# B&R Automation Studio project Soiled_PLC (part 13)

#### empty.var - Local variables
```iecst
(********************************************************************
 * COPYRIGHT --
 ********************************************************************
 * Program: pr
 * File: pr.var
 * Author: treamsbottom
 * Created: July 16, 2015
 ********************************************************************
 * Local variables of program pr
 ********************************************************************)
VAR
	mySeq : UINT;
	myIO : UINT;
	myZone : UINT;
	myRelLine : UINT;
	myBag : UINT;
	i_bagAtBuffer : BOOL;
	i_bagAtBufferOut : BOOL;
	i_bufferOutOpen : BOOL;
	o_openBuffer : BOOL;
	step : UINT;
	pls : BOOL;
	timerAlarm : TON_10ms;
END_VAR
VAR RETAIN
	lastStep : UINT;
END_VAR
VAR
	bufferSettleTime : UDINT;
	myOutBag : UINT;
	myBuffBag : UINT;
	myCan : UINT;
	alarm : REFERENCE TO Alm;
	bag : REFERENCE TO Bag_typ;
	bag_buff : REFERENCE TO Bag_typ;
	bag_out : REFERENCE TO Bag_typ;
	can : REFERENCE TO CAN_Vars;
	line_release : REFERENCE TO Line_Typ;
END_VAR
```

### Package Logical/BaseStandards/Incline - *Incline conveyor

- Standard_Sequence_Incline_ENG.docx (binary file, 206111 bytes)
### Program Logical/BaseStandards/Incline/ic (IEC, version 1.00.5) - *incline

#### ic.st - Implementation code
```iecst
(********************************************************************
 * COPYRIGHT --
 ********************************************************************
 * Program: ic
 * File: ic.st
 * Author: treamsbottom
 * Created: July 17, 2015
 ********************************************************************
 * Implementation of program Incline conveyor.
 ********************************************************************)
//V1.00.1 First Release
PROGRAM _INIT
//Configuration
mySeq					:= 15;		//Sequence number
myIO					:= 171; 	//Incline Conveyor IO module number
myIC					:= 1;		//Incline Conveyor Number
useRequest				:= FALSE; 	//Use the Request bit. Only use when working with x_1_point. otherwise use RequestRelease as the i_bagAtBuffer.
myBuffBag				:= 270;		//Ingoing Buffer bag number
myBag					:= 290;		//Incline bag number
myRelLine				:= 23;
myOutBag				:= Line[myRelLine].LastBag;	//Outgoing buffer bag number

myZone 					:= 0;
//Timer Values
bufferSettleTime		:= 300;  	// Time for bag to settle at buffer in.
moveUpInclineTime		:= 8;//>>IN SECONDS<< // Time to move bag up incline after closing stop.//Min of 4 to shut buffer stop....

alarm						ACCESS ADR(Alarm[mySeq]);
bag							ACCESS ADR(Bag[myBag]);
bag_buff					ACCESS ADR(Bag[myBuffBag]);
bag_out						ACCESS ADR(Bag[myOutBag]);
line_release				ACCESS ADR(Line[myRelLine]);
END_PROGRAM

PROGRAM _CYCLIC
//Inputs
i_paddleInPosition		:= X[myIO].X01;
i_bagAtBuffer			:= X[myIO].X03;
i_bagInIncline			:= X[myIO].X04;
i_BagReleased			:= FALSE;//X[myIO].X05;  //<--- Bag release trip- only to be used in special cases. Take when using tracked bags, as the next sequence will need to copy data into a transit position

i_bagAtBufferOut 		:= FALSE; // Any Single bag buffer out IO.
i_bufferOutOpen			:= FALSE;

//End of inputs.

o_openBuffer			:= FALSE;
o_runMotor				:= FALSE;

Request.IC[myIC] 		:= FALSE;
RequestRel.IC[myIC] 	:= FALSE;

IF (myBag = 0) THEN
	alarm.Bag	:= mySeq + 10000;
ELSE
	alarm.Bag	:= myBag;
END_IF;

alarm.Name 		:= 0;
alarm.Beacon		:= TRUE;
alarm.Extra		:= 0;
alarm.Time		:= 3000;

//Setup Sequence
step := D[900 + mySeq];
//Setup Pulse contact
pls := (step <> laststep);
laststep := step;

//Sequence
IF (step = 0) THEN
	//Disabled
END_IF;

//Run Incline until paddle in position
IF (step = 1) THEN
	o_runMotor := NOT i_paddleInPosition;
	IF i_paddleInPosition THEN
		D[900 + mySeq] := 2;
		Count[mySeq] := Count[mySeq] + 1;
	END_IF;
	IF NOT Std.HaltSysZone[myZone] THEN
		alarm.Name := ALM_SWITCH_FAULT;
	END_IF;
END_IF;

//Wait for at buffer
ton_10ms_SettledBuffer(IN:= i_bagAtBuffer, PT:= bufferSettleTime);
IF (step = 2) THEN
	IF NOT i_bagInIncline THEN
		IF useRequest THEN
			D[900 + mySeq] := 3;
		ELSE
			IF ton_10ms_SettledBuffer.Q THEN
				IF (myBuffBag > 0) THEN
					IF (bag_buff.Cat > 0) AND (bag.Cat = 0) THEN
						D[900 + mySeq] := 3;
					ELSIF (bag_buff.Cat = 0) THEN
						alarm.Name := ALM_BAG_DATA_ERROR;
						alarm.Bag := myBuffBag;
					ELSE
						alarm.Name := ALM_BAG_DATA_ERROR;
					END_IF;
				ELSE
					D[900 + mySeq] := 3;
				END_IF;
			ELSIF (myBuffBag > 0) AND (bag_buff.Cat > 0) THEN
				alarm.Name := ALM_BAG_NOT_SETTLED;
			END_IF;
		END_IF;
	ELSE
		alarm.Name := ALM_SWITCH_FAULT;
	END_IF;
END_IF;

//Open Buffer stop
IF (step = 3) THEN
	releaseValid := ((myBag = 0) OR ((bag.Cat = 0) AND (bag_buff.Cat > 0)));
	o_openBuffer	   := releaseValid AND NOT useRequest;
	Request.IC[myIC]  := releaseValid AND useRequest;
	IF i_bagInIncline AND releaseValid THEN
		IF (myBag > 0) THEN
			bag := bag_buff; //Clear empty buffer bag data if used
			bag_buff := Bag[0];
		END_IF;
		D[900 + mySeq] := 4;
	ELSIF (myBag > 0) THEN
		IF (bag.Cat > 0) THEN
			alarm.Name := ALM_BAG_DATA_ERROR;
			alarm.Time := 0;
		ELSIF (bag_buff.Cat = 0) THEN
			alarm.Name := ALM_BAG_DATA_ERROR;
			alarm.Bag := myBuffBag;
			alarm.Time := 0;
		ELSE
			alarm.Name  := ALM_BAG_NOT_ARRIVED;
		END_IF;
	ELSE
		alarm.Name  := ALM_BAG_NOT_ARRIVED;
	END_IF;
END_IF;

ton_10ms_SettledIncline(IN:= (step = 4), PT:= 300);
IF (step = 4) THEN
	o_openBuffer := NOT useRequest;
	IF ton_10ms_SettledIncline.Q THEN
		D[900 + mySeq] := 5;
	END_IF;
END_IF;

//Move Bag up incline
ctu_moveUpIncline(CU:=(step = 5) AND NOT Std.HaltSysZone[myZone] AND Std.Clock1s, RESET := (step <> 5), PV := moveUpInclineTime);
IF (step = 5) THEN
	o_openBuffer 	:= (ctu_moveUpIncline.CV <= 4) AND NOT useRequest;//Close buffer stop after 3 seconds running..
	o_runMotor 		:= TRUE;
	IF ctu_moveUpIncline.Q THEN
		D[900 + mySeq] := 6;
	ELSIF NOT Std.HaltSysZone[myZone] THEN
		alarm.Name := ALM_SWITCH_FAULT;
	END_IF;

END_IF;

//Check for line space.
IF (step = 6) THEN
	releaseValid := (NOT i_bagAtBufferOut AND NOT i_bufferOutOpen AND NOT i_BagReleased AND ((myBag = 0) OR ((bag.Cat > 0) AND (bag_out.Cat = 0))));
	IF (myRelLine > 0) THEN
		IF (line_release.Clear AND releaseValid) THEN
			C[myRelLine] := 0;
			D[900 + mySeq] := 7;
		END_IF;
		IF (line_release.Clear AND i_bagAtBufferOut) THEN
			alarm.Name := ALM_SWITCH_FAULT;
		ELSIF (myBag > 0) AND (bag.Cat = 0) THEN
			alarm.Name := ALM_BAG_DATA_ERROR;
			alarm.Time := 0;
		ELSIF line_release.Clear AND (myOutBag > 0) AND (bag_out.Cat > 0) THEN
			alarm.Name := ALM_BAG_DATA_ERROR;
			alarm.Bag := myOutBag;
			alarm.Time := 0;
		END_IF;
	ELSE
		RequestRel.IC[myIC] := releaseValid;
		IF EnableRel.IC[myIC] AND releaseValid THEN

			D[900 + mySeq] := 7;
		ELSIF (myBag > 0) AND (bag.Cat = 0) THEN
			alarm.Name := ALM_BAG_DATA_ERROR;
			alarm.Time := 0;
		ELSIF (myOutBag > 0) AND (bag_out.Cat > 0) THEN
			alarm.Name := ALM_BAG_DATA_ERROR;
			alarm.Bag := myOutBag;
			alarm.Time := 0;
		END_IF;
	END_IF;
	IF i_BagReleased THEN
		alarm.Name := ALM_SWITCH_FAULT;
		alarm.Time := 0;
	END_IF;
	releaseValid := 0; //Clear this as we are using it as a latch in line 7
END_IF;

//Run motor to release bag.
IF (step = 7) THEN
	IF (NOT i_bagAtBufferOut AND NOT i_bufferOutOpen AND ((myBag = 0) OR ((bag.Cat > 0) AND (bag_out.Cat = 0)))) THEN
		releaseValid := 1;
	END_IF;
	o_runMotor := releaseValid AND NOT Std.HaltSysZone[myZone];
	IF releaseValid THEN
		IF (myBag = 0) THEN
			IF (myRelLine > 0) THEN
				IF line_release.Trip THEN
					D[900 + mySeq] := 1;
				END_IF;
			ELSE
				IF NOT EnableRel.IC[myIC] OR i_BagReleased THEN
					D[900 + mySeq] := 1;
				END_IF;
			END_IF;
			IF NOT Std.HaltSysZone[myZone] THEN
				alarm.Name := ALM_BAG_NOT_RELEASED;
			END_IF;
		ELSE//Use tracking
			IF (myRelLine > 0) THEN
				IF line_release.Trip THEN
					bag_out := bag;
					bag := Bag[0];
					D[900 + mySeq] := 1;
				END_IF;
			ELSE
				IF (i_BagReleased OR NOT EnableRel.IC[myIC]) AND (bag.Cat = 0)  THEN // Make sure data is copied out by enabling sequence.
					D[900 + mySeq] := 1;
				ELSIF NOT EnableRel.IC[myIC] AND (bag.Cat > 0) THEN
					alarm.Name := ALM_BAG_DATA_ERROR;
				END_IF;
			END_IF;
		END_IF;
	ELSIF i_bagAtBufferOut OR i_bufferOutOpen THEN
			alarm.Name := ALM_SWITCH_FAULT;
			alarm.Time := 0;
	ELSIF (myBag > 0) THEN
		IF (bag.Cat = 0) THEN
			alarm.Name := ALM_BAG_DATA_ERROR;
			alarm.Time := 0;
		ELSIF (bag_out.Cat > 0) THEN
			alarm.Name := ALM_BAG_DATA_ERROR;
			alarm.Bag := myOutBag;
			alarm.Time := 0;
		END_IF;
	END_IF;
END_IF;

//-----------------------------------
//PLC Outputs - adjust TO suit system
//-----------------------------------

Y[7].Y01	:= o_runMotor;
Y[myIO].Y06 := o_openBuffer;

//Alarms
timerAlarm(IN := NOT pls AND (alarm.Name > 0),PT:= alarm.Time);

alarm.On 	:= timerAlarm.Q;
alarm.ET 	:= timerAlarm.ET;;

END_PROGRAM
```

### Package Logical/BaseStandards/LoadingUnit - *Loading Unit

- Standard_Sequence_IoadingUnit_ENG.docx (binary file, 208000 bytes)
### Program Logical/BaseStandards/LoadingUnit/lu (IEC, version 1.01.1) - *Loading Unit

#### lu.var - Local variables
```iecst
(********************************************************************
 * COPYRIGHT --
 ********************************************************************
 * Program: lu
 * File: lu.var
 * Author: treamsbottom
 * Created: July 17, 2015
 ********************************************************************
 * Local variables of program lu
 ********************************************************************)
VAR
	useRequest : BOOL;
	useCompressor : BOOL;
	ton_10ms_SteadyDown : TON_10ms;
	ton_10ms_SettleInLU : TON_10ms;
	timerAlarm : TON_10ms;
	switchFault : BOOL;
	step : UINT;
	releaseValid : BOOL;
	pls : BOOL;
	o_steadyCylinders : BOOL;
	o_openBuffer : BOOL;
	o_openBackStop : BOOL;
	o_moveCompressorDown : BOOL;
	myZone : UINT;
	mySeq : UINT;
	myRelLine : UINT;
	myOutBag : UINT;
	myLU : UINT;
	myIO : UINT;
	myBuffBag : UINT;
	myBag : UINT;
	lu_Enabled : BOOL;
END_VAR
VAR RETAIN
	lastStep : UINT;
END_VAR
VAR
	i_compressorAtTop : ARRAY[0..2] OF BOOL;
	i_compress : BOOL;
	i_bufferOutOpen : BOOL;
	i_bagInLoadingUnit : BOOL;
	i_bagFrontPast : BOOL;
	i_bagAtBufferOut : BOOL;
	i_bagAtBuffer : BOOL;
	compressorUp : BOOL;
	compress : BOOL;
	bufferSettleTime : UINT;
	myReportStn : UINT;
	myBelt : UINT;
	myCan : UINT;
	unloadFinished : BOOL;
	ton_10ms_LuClear : TON_10ms;
	ton_10ms_SettledBuffer : TON_10ms;
	ton_10ms_CompressCheck : TON_10ms;
	ton_10ms_CompressDown : TON_10ms;
	ton_10ms_CompressorCheck : TON_10ms;
	myPrg : USINT;
	myCat : UDINT;
	myCus : UDINT;
	myWgt : UINT;
	myMis : UDINT;
	alarm : REFERENCE TO Alm;
	bag : REFERENCE TO Bag_typ;
	bag_out : REFERENCE TO Bag_typ;
	bag_buff : REFERENCE TO Bag_typ;
	can : REFERENCE TO CAN_Vars;
	line_release : REFERENCE TO Line_Typ;
END_VAR
```

### lu.st - Implementation code
```iecst
(********************************************************************
 * COPYRIGHT --
 ********************************************************************
 * Program: lu
 * File: lu.st
 * Author: treamsbottom
 * Created: July 17, 2015
 ********************************************************************
 * Implementation of program lu
 ********************************************************************)
//V1.00.1 First Release
PROGRAM _INIT
//Configuration
mySeq						:= 1;	//Sequence number
myIO						:= 21;	//First IO Block
myLU						:= 1;	// Loading unit number
myZone						:= 0;	// Safety Zone
myRelLine					:= 22; 	// Release Line - Set to 0 to Request Release
myBag						:= 255; //Buffer Bag
myBuffBag					:= 0; 	// Tracking Empty bag in...
useRequest					:= FALSE; 	//Use the Request bit. Only use when working with x_1_point. otherwise use RequestRelease as the i_bagAtBuffer.
bufferSettleTime			:= 300; // Time for bag to settle in buffer

useCompressor				:= FALSE;
myReportStn					:= 0;//myLU// Set Station index for reports. 0 = no report write.

myBelt						:= 1;	// Set if loaded by a belt
myCan						:= 0;	// Set if using Kanlink...

myOutBag					:= Line[myRelLine].LastBag;

alarm						ACCESS ADR(Alarm[mySeq]);
bag							ACCESS ADR(Bag[myBag]);
bag_buff					ACCESS ADR(Bag[myBuffBag]);
bag_out						ACCESS ADR(Bag[myOutBag]);
can							ACCESS ADR(CAN[myCan]);
line_release				ACCESS ADR(Line[myRelLine]);

END_PROGRAM

PROGRAM _CYCLIC
//Inputs
i_bagAtBuffer			:= X[myIO].X01;
i_bagFrontPast			:= X[myIO].X02;
i_bagInLoadingUnit		:= X[myIO].X03;
i_compressorAtTop[1]	:= TRUE; // Set to TRUE if there is no compressor
i_compressorAtTop[2]	:= TRUE;
i_compress				:= FALSE;

i_bagAtBufferOut 		:= FALSE; // Any Single bag buffer out IO.
i_bufferOutOpen			:= FALSE;

o_openBuffer			:= FALSE;
o_steadyCylinders		:= FALSE;
o_openBackStop	 		:= FALSE;
o_moveCompressorDown	:= FALSE;

Request.LU[myLU]		:= FALSE;
RequestRel.LU[myLU]		:= FALSE;
IF (myBelt > 0) THEN
	EnableRel.TransferBelt[myBelt] := FALSE;
END_IF;
IF (myCan > 0) THEN
	can.ReadyToLoad := FALSE;
END_IF

IF (myBag = 0) THEN
	alarm.Bag	:= mySeq + 10000;
ELSE
	alarm.Bag	:= myBag;
END_IF;

alarm.Name 		:= 0;
alarm.Beacon		:= TRUE;
alarm.Extra		:= 0;
alarm.Time		:= 3000;

//Setup Sequence
step := D[900 + mySeq];
//Setup Pulse contact
pls := (step <> lastStep);
lastStep := step;

//Get BagID
IF (bag.Cat > 0) AND (bag.Bid = 0) AND (BidStn > 0) THEN
	bag.Bid := BidStn;
	BidStn := 0;
END_IF;

//Sequence
IF (step = 0) THEN
	//Disabled
END_IF;

lu_Enabled	:= ((D[mySeq] > 0) AND NOT Std.HaltSysZone[myZone]);

//Check loading unit is clear.
switchFault 	:= (i_bagFrontPast OR i_bagInLoadingUnit);
compressorUp 	:= (i_compressorAtTop[1] AND i_compressorAtTop[2]);
ton_10ms_LuClear(IN:= compressorUp AND NOT switchFault,PT:= 200);
IF (step = 1) THEN
	IF (ton_10ms_LuClear.Q AND lu_Enabled) THEN
		D[900 + mySeq] := 2;
		Count[mySeq] := Count[mySeq] + 1;
	END_IF;
	IF (switchFault OR NOT compressorUp) THEN
		alarm.Name := ALM_SWITCH_FAULT;
	END_IF;
END_IF;

// Step 2 - Wait for bag at buffer if used
ton_10ms_SettledBuffer(IN:= i_bagAtBuffer, PT:= bufferSettleTime);
IF (step = 2) THEN
	IF useRequest THEN
		D[900 + mySeq] := 3;
	ELSE
		IF ton_10ms_SettledBuffer.Q THEN
			IF (myBuffBag > 0) THEN
				IF (bag_buff.Cat > 0) AND (bag.Cat = 0) THEN
					D[900 + mySeq] := 3;
				ELSIF (bag_buff.Cat = 0) THEN
					alarm.Name := ALM_BAG_DATA_ERROR;
					alarm.Bag := myBuffBag;
				ELSE
					alarm.Name := ALM_BAG_DATA_ERROR;
				END_IF;
			ELSE
				D[900 + mySeq] := 3;
			END_IF;
		ELSIF (myBuffBag > 0) AND (bag_buff.Cat > 0) THEN
			alarm.Name := ALM_BAG_NOT_SETTLED;
		END_IF;
	END_IF;
END_IF;

//Open buffer stop / Request bag
IF (step = 3) THEN
	releaseValid := ((myBuffBag = 0) OR ((bag.Cat = 0) AND (bag_buff.Cat > 0)));
	o_openBuffer := releaseValid AND NOT useRequest;
	o_openBackStop := TRUE;
	Request.LU[myLU]  := releaseValid AND useRequest;
	IF i_bagFrontPast AND releaseValid THEN
		IF (myBuffBag > 0) THEN
			bag := bag_buff; //Clear empty buffer bag data if used
			bag_buff := Bag[0];
		END_IF;
		D[900 + mySeq] := 4;
	ELSIF (myBuffBag > 0) THEN
		IF (bag.Cat > 0) THEN
			alarm.Name := ALM_BAG_DATA_ERROR;
			alarm.Time := 0;
		ELSIF (bag_buff.Cat = 0) THEN
			alarm.Name := ALM_BAG_DATA_ERROR;
			alarm.Bag := myBuffBag;
			alarm.Time := 0;
		ELSE
			alarm.Name  := ALM_BAG_NOT_ARRIVED;
		END_IF;
	ELSE
		alarm.Name  := ALM_BAG_NOT_ARRIVED;
	END_IF;
END_IF;

//Step 4 - Bag settles in loading unit
ton_10ms_SettleInLU(IN:= i_bagInLoadingUnit,PT:= 300);
IF (step = 4) THEN
	IF ton_10ms_SettleInLU.Q THEN
		D[900 + mySeq] := 5;
	END_IF;
	alarm.Name := ALM_BAG_NOT_SETTLED;
END_IF;

//Steady cylinders on from steps 5 - 8
o_steadyCylinders := ((step >= 5) AND (step <= 8));

//Move Steady Cylinders down and check bag data
ton_10ms_SteadyDown(IN:= (step = 5), PT:= 200);
IF (step = 5) THEN
	IF ton_10ms_SteadyDown.Q  THEN
		IF (myBuffBag = 0) THEN
			IF (bag.Cat = 0) THEN
				D[900 + mySeq] := 6;
			ELSE
				alarm.Name := ALM_BAG_DATA_ERROR;
				alarm.Time := 0;
			END_IF;
		ELSE
			IF (bag.Cat = Std.MaxCats) THEN
				D[900 + mySeq] := 6;
			ELSE
				alarm.Name := ALM_BAG_DATA_ERROR;
				alarm.Time := 0;
			END_IF;
		END_IF;
	END_IF;
END_IF;

//Step 6 Wait for bag to be loaded..
IF (step = 6) THEN
	EnableRel.TransferBelt[myBelt] 	:= (myBelt > 0);
	IF (myCan > 0) THEN// Kanlink interface.
		can.ReadyToLoad 		:= NOT unloadFinished;
		IF (can.Category > 0) AND NOT unloadFinished THEN
			myPrg := UINT_TO_USINT(can.Program);
			myCat := can.Category;
			myCus := can.Customer;
			myWgt := can.Weight;
			myMis := can.BatchID;
		END_IF;
		// Get Program code
		IF ((myPrg = 0) AND (myCat > 0) AND (D32[100 + 20 * (myLU - 1)] <> myCat)) THEN
			D32[100 + 20 * (myLU - 1)] := myCat;
		ELSIF (D32[101 + 20 * (myLU - 1)] = myCat) THEN
			myPrg := UDINT_TO_USINT(D32[102 + 20 * (myLU - 1)]);
		END_IF;
		IF can.UnloadFinished THEN
			unloadFinished := TRUE;
		END_IF;
		IF (unloadFinished AND (myCat > 0) AND (myPrg > 0)) THEN
			bag.Prg := myPrg;
			bag.Cat := myCat;
			bag.Cus := myCus;
			bag.Wgt := myWgt;
			bag.Mis := myMis;
		END_IF;
	END_IF;

	IF (bag.Cat > 0) AND (bag.Prg > 0) AND ((bag.Cat <> Std.MaxCats) OR (myBuffBag = 0)) THEN
		IF (myReportStn > 0) THEN
			IF (ReportLoading[myReportStn].Cat = 0) THEN
				ReportLoading[myReportStn].Prg := bag.Prg;
				ReportLoading[myReportStn].Cat := bag.Cat;
				ReportLoading[myReportStn].Cus := bag.Cus;
				ReportLoading[myReportStn].Wgt := bag.Wgt;
				ReportLoading[myReportStn].Cnt := 0;
				ReportLoading[myReportStn].Stn := myReportStn;
				ReportLoading[myReportStn].Mcn := 0;
				ReportLoading[myReportStn].Bid := bag.Mis;
				D[900 + mySeq] := 7;
			END_IF;
		ELSE
			D[900 + mySeq] := 7;
		END_IF;
	ELSIF (myCan > 0) AND unloadFinished THEN
		alarm.Name := ALM_BAG_DATA_ERROR;
	END_IF;
ELSE
	D32[100 + 20 * (myLU - 1)] := 0;
	unloadFinished := FALSE;
	can.ReadyToLoad := FALSE;
	can.Program := 0;
	can.Category := 0;
	can.Customer := 0;
	can.Weight := 0;
	can.BatchID := 0;
END_IF;

//Step 7 Check If compression is required
ton_10ms_CompressCheck(IN:=(step = 7),PT:= 30);
IF (step = 7) THEN
	IF useCompressor THEN
		IF i_compress THEN
			compress := TRUE;
		END_IF;
		IF ton_10ms_CompressCheck.Q THEN
			IF compress THEN
				D[900 + mySeq] := 8; // Compress
			ELSE
				D[900 + mySeq] := 9;	// Check compressor is OK
			END_IF;
		END_IF;
	ELSE
		D[900 + mySeq] := 9;
	END_IF;
ELSE
	compress := FALSE;
END_IF;

//Step 8 move linen compressor down.
ton_10ms_CompressDown(IN:=(step = 8),PT:= 500);
IF (step = 8) THEN
	IF useCompressor THEN
		IF ton_10ms_CompressDown.Q THEN
			D[900 + mySeq] := 9;
		END_IF;
	ELSE
		D[900 + mySeq] := 9;
	END_IF;
END_IF;

//step 9 check compressor status
ton_10ms_CompressorCheck(IN:=((i_compressorAtTop[1] AND i_compressorAtTop[2]) OR NOT useCompressor),PT:= 200);
IF (step = 9) THEN
	IF ton_10ms_CompressorCheck.Q  AND NOT Std.HaltSysZone[myZone] THEN
		D[900 + mySeq] := 10;
	END_IF;
	alarm.Name := ALM_SWITCH_FAULT;
END_IF;

//Check for line space.
IF (step = 10) THEN
	releaseValid := (NOT i_bagAtBufferOut AND NOT i_bufferOutOpen AND (bag.Cat > 0) AND (bag_out.Cat = 0));
	IF NOT Std.HaltSysZone[myZone] THEN
		IF (myRelLine > 0) THEN
			IF (line_release.Clear AND releaseValid) THEN
				C[myRelLine] := 0;
				D[900 + mySeq] := 11;
			END_IF;
			IF (line_release.Clear AND i_bagAtBufferOut) THEN
				alarm.Name := ALM_SWITCH_FAULT;
			ELSIF (bag.Cat = 0) THEN
				alarm.Name := ALM_BAG_DATA_ERROR;
				alarm.Time := 0;
			ELSIF line_release.Clear AND (bag_out.Cat > 0) THEN
				alarm.Name := ALM_BAG_DATA_ERROR;
				alarm.Bag := myOutBag;
				alarm.Time := 0;
			END_IF;
		ELSE
			RequestRel.LU[myLU] := releaseValid;
			IF EnableRel.LU[myLU] AND releaseValid THEN
				D[900 + mySeq] := 11;
			ELSIF (myBag > 0) AND (bag.Cat = 0) THEN
				alarm.Name := ALM_BAG_DATA_ERROR;
				alarm.Time := 0;
			ELSIF (myOutBag > 0) AND (bag_out.Cat > 0) THEN
				alarm.Name := ALM_BAG_DATA_ERROR;
				alarm.Bag := myOutBag;
				alarm.Time := 0;
			END_IF;
		END_IF;
	END_IF;
END_IF;

//Release bag.
IF (step = 11) THEN
	releaseValid 	:= (NOT i_bagAtBufferOut AND NOT i_bufferOutOpen AND (bag.Cat > 0) AND (bag_out.Cat = 0));
	o_openBackStop := releaseValid;
	IF releaseValid THEN
		IF (myRelLine > 0) THEN
			IF line_release.Trip THEN
				bag_out := bag;
				bag := Bag[0];
				D[900 + mySeq] := 1;
			END_IF;
		ELSE
			IF NOT EnableRel.LU[myLU] AND (bag.Cat = 0) THEN // Make sure data is copied out by enabling sequence.
				D[900 + mySeq] := 1;
			ELSIF NOT EnableRel.LU[myLU] AND (bag.Cat > 0) THEN
				alarm.Name := ALM_BAG_DATA_ERROR;
			END_IF;
		END_IF;
	ELSIF i_bagAtBufferOut OR i_bufferOutOpen THEN
		alarm.Name := ALM_SWITCH_FAULT;
		alarm.Time := 0;
	ELSIF (bag.Cat = 0) THEN
		alarm.Name := ALM_BAG_DATA_ERROR;
		alarm.Time := 0;
	ELSIF (bag_out.Cat > 0) THEN
		alarm.Name := ALM_BAG_DATA_ERROR;
		alarm.Bag := myOutBag;
		alarm.Time := 0;
	END_IF;
END_IF;

//-----------------------------------
//PLC Outputs - adjust TO suit system
//-----------------------------------

Y[myIO].Y05 		:= o_openBuffer;
Y[myIO].Y06 		:= o_openBackStop;
Y[myIO].Y07 		:= o_steadyCylinders;
//Y[myIO + 1].Y05 	:= o_moveCompressorDown;
//Y[myIO + 1].Y06 	:= o_moveCompressorDown;
Y[myIO + 1].Y07 	:= o_steadyCylinders; //Elephants foot

//Alarms
timerAlarm(IN := NOT pls AND (alarm.Name > 0),PT:= alarm.Time);

alarm.On 	:= timerAlarm.Q;
alarm.ET 	:= timerAlarm.ET;

END_PROGRAM
```

### Package Logical/BaseStandards/On_Offgoing - *Old style on and offgoing points

- SequenceExample.doc (binary file, 73216 bytes)
### Program Logical/BaseStandards/On_Offgoing/x_pn (IEC) - *Ongoing Sequence

#### x_pn.ab
```automation-basic
PROGRAM _CYCLIC

;--------------------------------------
;Sequence 4 - Ongoing To Storage D[900 + mySeq]
;--------------------------------------

;--------------------------------------------------------------------------------
;Revision 1.00 06/11/2009 D.J. First Issue - Automatic Line Allocation with Areas
;--------------------------------------------------------------------------------
mySeq 			= 4
myZone 			= 0
myTransitBag	= 208
myStartStop		= 100

IF (myStartStop >= 100) THEN
	myStartStop = myStartStop + 7600
ENDIF

;Inputs
OnGoingEnable 		= ((D[mySeq] > 0) AND NOT Std.HaltSysZone[myZone])

I_BagatBuffer[1]		= X[221].X02
I_BagatBuffer[2]		= FALSE
I_BagatBuffer[3]		= FALSE
I_BagatBuffer[4]		= FALSE

O_Reset 		  		= FALSE
O_OpenSelect[1]			= FALSE
O_OpenSelect[2]			= FALSE
O_OpenSelect[3]			= FALSE
O_OpenSelect[4]			= FALSE

O_OpenBuffer[1]			= FALSE
O_OpenBuffer[2]			= FALSE
O_OpenBuffer[3]			= FALSE
O_OpenBuffer[4]			= FALSE

MaxBuffers 			= 1 	;Set Max Buffers to search
MinLine				= 1 	;Set First Storage Line
MaxLine				= 10		;Set Last Storage Line
MaxDepth			= 7    ;Capacity of the longest line - used in search

Alarm[mySeq].Name 		= 0
Alarm[mySeq].Bag		= myTransitBag
Alarm[mySeq].Beacon		= TRUE
Alarm[mySeq].Extra	 	= 0
Alarm[mySeq].Time		= 6000

;Setup Sequence
;--------------
STEP = D[900 + mySeq]
;Setup Pulse contact
PLS = (STEP <> LASTSTEP)
LASTSTEP = STEP

;Step 0 - Disabled
IF (STEP = 0) THEN
	;Disabled
ENDIF

;Step 1 - Reset Ongoing Points
TON_10ms((STEP = 1),300,ResetPoints,ResetPointsET)
IF (STEP = 1) THEN
	Dest  	= 0
	Buff 	= 0
	O_Reset = TRUE
	IF (ResetPoints AND OnGoingEnable) THEN
		D[900 + mySeq] = 2
	ENDIF
ENDIF

;Bag Settles at each buffer
TON_10ms(I_BagatBuffer[1],300,SettledBuffer[1],SettledBufferET[1])
;TON_10ms(I_BagatBuffer[2],300,SettledBuffer[2],SettledBufferET[2])
;TON_10ms(I_BagatBuffer[3],300,SettledBuffer[3],SettledBufferET[3])

BufferBagNum[1]	    = 211
;BufferBagNum[2]	= 161
;BufferBagNum[3]	= myTransitBag

;Step 2 - Search for a valid Bag at one of the buffers
IF (STEP = 2) THEN

	Buff 	= 0
	Dest 	= 0

	IF OnGoingEnable THEN

		Alarm[mySeq].Name 	= almNoAlarm

		;Search only 1 buffer bag per scan/task
		Buffer = Buffer + 1
		IF Buffer > MaxBuffers THEN
			Buffer = 1
		ENDIF
		;Set Test Value for Monitoring
		IF TestBuffer > 0 THEN
			Buffer = TestBuffer
		ENDIF

		BufferBag		= BufferBagNum[Buffer]
		BufferSettled 	= SettledBuffer[Buffer]
		BufferPrg 		= Bag[BufferBag].Prg
		BufferCat		= Bag[BufferBag].Cat
		BufferCus		= Bag[BufferBag].Cus
		BufferDst 		= Bag[BufferBag].Dst

		IF (BufferSettled AND (BufferCat > 0) AND (BufferPrg > 0) AND (BufferPrg <= Std.MaxProg) AND (OnGoingEnable)) THEN

			;Manual Destination has been set?
			IF (BufferDst > 0) THEN

				n = BufferDst
				IF ((n >= MinLine) AND (n <= MaxLine) AND (Line[n].Space > 0) AND Line[n].Clear) THEN
					Dest 	= n
					Buff 	= Buffer
					D[900 + mySeq] 	= 3
				ELSE
					Alarm[mySeq].Name 	= almDestinationNotValid
					Alarm[mySeq].Bag	= BufferBag
				ENDIF

			ELSE IF Std.AutoLineAllocation THEN ;/BufferDst > 0

				;Search Each Storage Area
				AreaChoice[1] = D[3000 + BufferPrg]
				AreaChoice[2] = D[3100 + BufferPrg]
				AreaChoice[3] = D[3200 + BufferPrg]
				AreaChoice[4] = D[3300 + BufferPrg]

				LOOP Area = 1 TO 4 DO

					AreaStartLine 	= D[250 + AreaChoice[Area]]
					AreaEndLine 	= D[270 + AreaChoice[Area]]
					AreaValid		= ((AreaStartLine > 0) AND (AreaEndLine > 0) AND (AreaEndLine >= AreaStartLine))
					IF AreaValid THEN

						;Search for a line with the same program
						;---------------------------------------
						LOOP myLine = AreaStartLine TO AreaEndLine DO
							myLineValid = ((myLine >= MinLine) AND (myLine <= MaxLine))
							myLineUsed	= (D[myStartStop + myLine] > 0) ;Start / Stop On
							IF myLineValid AND myLineUsed THEN
								n 			= myLine
								SearchBag 	= (Line[n].LastBag - Line[n].Space)
								IF ((SearchBag >= Line[n].FirstBag) AND (Bag[SearchBag].Prg = BufferPrg) AND (Line[n].Space > 0) AND Line[n].Clear) THEN
									;Found line with a matching program
									Dest 	= n
								ENDIF ;/SearchBag
							ENDIF ;/myLineValid
							EXITIF (Dest <> 0)
						ENDLOOP ;/myLine loop

						;Search for an empty line
						;------------------------
						IF (Dest = 0) THEN
							LOOP myLine = AreaStartLine TO AreaEndLine DO
								myLineValid = ((myLine >= MinLine) AND (myLine <= MaxLine))
								myLineUsed	= (D[myStartStop + myLine] > 0) ;Start / Stop On
								IF myLineValid AND myLineUsed THEN
									n 			= myLine
									SearchBag 	= (Line[n].FirstBag)
									IF ((Bag[SearchBag].Prg = 0) AND (Line[n].Space > 0) AND Line[n].Clear) THEN
										;Found line with a matching program
										Dest 	= n
									ENDIF ;/SearchBag
								ENDIF ;/myLineValid
							EXITIF (Dest <> 0)
							ENDLOOP ;/myLine loop
						ENDIF ;/Dest = 0

						;Search for a line that already contains a bag with the same program starting at the back
						;----------------------------------------------------------------------------------------
						IF (Dest = 0) THEN
							LOOP myDepth = (MaxDepth - 2) DOWNTO 0 DO ;Don't search the last bag as the line would already be full!!
								LOOP myLine = AreaStartLine TO AreaEndLine DO
									myLineValid = ((myLine >= MinLine) AND (myLine <= MaxLine))
									myLineUsed	= (D[myStartStop + myLine] > 0) ;Start / Stop On
									IF myLineValid AND myLineUsed THEN
										n 			= myLine
										SearchBag 	= (Line[n].FirstBag + myDepth)
										IF ((Bag[SearchBag].Prg = BufferPrg) AND (Line[n].Space > 0) AND Line[n].Clear) THEN
											;Found line with a matching program
											FoundDepth 	= myDepth
											Dest 		= n
										ENDIF ;/SearchBag
									ENDIF ;/myLineValid
									EXITIF (Dest <> 0)
								ENDLOOP ;/myLine loop
								EXITIF (Dest <> 0)
							ENDLOOP ;/myDepgh
						ENDIF ;/Dest = 0

						;Search for line with the most space
						;-----------------------------------
						IF (Dest = 0) THEN
							mySpace = 0
							myFound	= 0
							LOOP myLine = AreaStartLine TO AreaEndLine DO
								myLineValid = ((myLine >= MinLine) AND (myLine <= MaxLine))
								myLineUsed	= (D[myStartStop + myLine] > 0) ;Start / Stop On
								IF myLineValid AND myLineUsed THEN
									n 			= myLine
									SearchBag 	= (Line[n].LastBag)
									IF ((Bag[SearchBag].Prg = 0) AND (Line[n].Space > mySpace) AND Line[n].Clear) THEN
										;Found line with a matching program
										myFound	= n
										mySpace = Line[n].Space
									ENDIF ;/SearchBag
								ENDIF ;/myLineValid
							ENDLOOP ;/myLine loop

							IF (myFound > 0) THEN
								Dest 	= myFound
							ENDIF

						ENDIF ;/Dest = 0

					ENDIF ;/Area Valid
					EXITIF (Dest <> 0)
				ENDLOOP ;/Area Loop

			ENDIF ;/BufferDst > 0

			;Destination line found!!
			IF (Dest <> 0) THEN
				Buff = Buffer
				IF (Bag[myTransitBag].Cat = 0) AND (Bag[BufferBagNum[Buff]].Cat > 0) THEN ;Bag in Transit
					Bag[BufferBagNum[Buff]].Dst = USINT(Dest)
					Bag[myTransitBag]	= Bag[BufferBagNum[Buff]]
					Bag[BufferBagNum[Buff]]	 	= Bag[0]
					C[Dest] = 0
					D[900 + mySeq] 	= 3 ; Open buffer
				ENDIF
			ELSE
				;Storage full!!
				;Do Nothing? Alarm?
				;Other Area?
			ENDIF

		ENDIF ;/BagSettled

		;Buffer Alarms
		IF (BufferPrg > 0) AND NOT BufferSettled THEN
			Alarm[mySeq].Name 	= almBagNotAtProx
			Alarm[mySeq].Bag	= BufferBag
		ELSE IF (BufferPrg = 0) AND BufferSettled THEN
			Alarm[mySeq].Name 	= almBagNotShownOnScreen
			Alarm[mySeq].Bag	= BufferBag
		ENDIF
	ENDIF
ENDIF

;Clear Line Selections
LOOP n = 1 TO Std.MaxLines DO
	LineSelect[n] = FALSE
ENDLOOP

;Step 3 - Select line / open buffer stop
IF (STEP = 3) THEN
	LineSelect[Dest] 	= TRUE
	O_OpenBuffer[Buff] = TRUE
	;Bag arrived on selected line
	IF Line[Dest].Trip THEN
		D32[498] 					= Bag[myTransitBag].Cus	;Set Customer for Customer FIFO
		Bag[myTransitBag].Dst 		= 0 		    ;Clear Destination
		Bag[Line[Dest].LastBag] 	= Bag[myTransitBag]
		Bag[myTransitBag] 			= Bag[0]
		D[900 + mySeq] 				= 1
	ENDIF
	Alarm[mySeq].Name = almBagNotArrived
ENDIF

;Alarms
TimerAlarm.IN = NOT PLS AND (Alarm[mySeq].Name > 0) AND (AlarmOld = Alarm[mySeq].Name)
TimerAlarm.PT = Alarm[mySeq].Time
TimerAlarm FUB TON_10ms()
Alarm[mySeq].On = TimerAlarm.Q
Alarm[mySeq].ET = TimerAlarm.ET

AlarmOld = Alarm[mySeq].Name ;Need to ensure alarm changes as may be multiple alarms on step 2

Y[221].Y06 = O_OpenBuffer[1]

;Outputs
Y[51].Y08 = O_Reset
Y[52].Y07 = O_Reset
Y[53].Y07 = O_Reset
Y[53].Y08 = O_Reset
Y[54].Y07 = O_Reset
Y[54].Y08 = O_Reset
Y[55].Y07 = O_Reset
Y[55].Y08 = O_Reset
Y[56].Y07 = O_Reset

Y[51].Y06 = LineSelect[2]
Y[52].Y05 = LineSelect[3]
Y[53].Y05 = LineSelect[4]
Y[53].Y06 = LineSelect[5]
Y[54].Y05 = LineSelect[6]
Y[54].Y06 = LineSelect[7]
Y[55].Y05 = LineSelect[8]
Y[55].Y06 = LineSelect[9]
Y[56].Y05 = LineSelect[10]

END_PROGRAM
```

### Program Logical/BaseStandards/On_Offgoing/x_pf (IEC) - *Offgoing Sequence

#### pf1.var
```iecst
VAR RETAIN
	LASTSTEP : UINT;
	SelectedBuffer : USINT;
	Destination : UINT;
	FoundLine : UINT;
END_VAR
VAR
	x : UINT;
	Line14_Valid : BOOL;
	LongestLine : UINT;
	O_Select : ARRAY[0..22] OF BOOL;
	LongestSTime : UINT;
	LineInList : ARRAY[0..98] OF BOOL;
	mySeq : UINT;
	RecircSpaces : UINT;
	O_Reset3way : BOOL;
	r : UINT;
	myRelLine : UINT;
	SettleTime : UINT;
	TransitBag : UINT;
	RecircValid : BOOL;
	TimerAlarm : TON_10ms;
	SDC6_Valid : BOOL;
	SDC5_Valid : BOOL;
	SDC7_Valid : BOOL;
	TestAtStop : BOOL;
	STEP : UINT;
	SDC3_Valid : BOOL;
	SearchDest : UINT;
	SDC4_Valid : BOOL;
	I_InclineBufferStopOpen : BOOL;
	ResetPointsET : TIME;
	ResetPoints : BOOL;
	OffGoingEnable : BOOL;
	SDC1_Valid : BOOL;
	SDC2_Valid : BOOL;
	PLS : BOOL;
	O_SDCBufferOpen : ARRAY[0..4] OF BOOL;
	O_Reset : BOOL;
	MaxLine : UINT;
	n : UINT;
	MinLine : UINT;
	BufferBag : ARRAY[0..9] OF UINT;
	LineSelect : ARRAY[0..30] OF BOOL;
	MaxBuffers : UINT;
	I_SDCBagAtBuffer : ARRAY[0..4] OF BOOL;
	I_BagAtIncline : BOOL;
	IncSettle : BOOL;
	LineSettle : ARRAY[0..30] OF BOOL;
	BestTime : UINT;
	BufferClear : ARRAY[0..9] OF BOOL;
	AlarmBagNotProx : BOOL;
	I_BagAtStop : ARRAY[0..30] OF BOOL;
	BagSettledTime : ARRAY[0..30] OF UINT;
	myZone : UINT;
END_VAR
```

#### pf1.ab
```automation-basic
PROGRAM _CYCLIC

;----------------------------------------
;Sequence 5 - SPF1 Offgoing Points D[900+mySeq]
;----------------------------------------

;Inputs
;------
mySeq			= 5
myRelLine 		= 26
TransitBag 		= 207
myZone			= 0

OffGoingEnable 		= ((D[mySeq] > 0) AND NOT Std.HaltSysZone[myZone])

I_SDCBagAtBuffer[1] = X[213].X01 ;Bag In Discharger
I_SDCBagAtBuffer[2] = FALSE ;Use for single bag buffer
I_SDCBagAtBuffer[3] = FALSE ;X[6].X13 ;Use for single bag buffer
I_SDCBagAtBuffer[4] = FALSE ;X[6].X13 ;Use for single bag buffer

O_SDCBufferOpen[1]  = Y[213].Y05 ;Use for single bag buffer
O_SDCBufferOpen[2]  = FALSE ;Use for single bag buffer
O_SDCBufferOpen[3]  = FALSE ;Y[6].Y16 ;Use for single bag buffer
O_SDCBufferOpen[4]  = FALSE ;Y[6].Y16 ;Use for single bag buffer

I_BagAtStop[1]	 	= X[71].X01 OR TestAtStop
I_BagAtStop[2] 		= X[71].X02 OR TestAtStop
I_BagAtStop[3] 		= X[72].X01 OR TestAtStop
I_BagAtStop[4] 		= X[72].X02 OR TestAtStop
I_BagAtStop[5] 		= X[73].X01 OR TestAtStop
I_BagAtStop[6]	 	= X[73].X02 OR TestAtStop
I_BagAtStop[7] 		= X[74].X01 OR TestAtStop
I_BagAtStop[8] 		= X[74].X02 OR TestAtStop
I_BagAtStop[9] 		= X[75].X01 OR TestAtStop
I_BagAtStop[10] 	= X[75].X02 OR TestAtStop

O_Reset 			= FALSE

;Buffer line configuration
;-------------------------
MaxBuffers			= 1
MinLine				= 1
MaxLine				= 10

BufferBag[1]		= 251 ;Last buffer bag number
;BufferBag[2]		= 373;Last buffer bag number
;BufferBag[3]		= 383 ;Last buffer bag number CDC3
;BufferBag[4]		= 192 ;Last buffer bag number CDC4
;BufferBag[5]		= 155 ;Last buffer bag number CDC 5
;BufferBag[6]		= 658 ;Last buffer bag number
;BufferBag[7]		= 664 ;Last buffer bag number
;RecircSpaces  		=(Line[20].Space + Line[24].Space + (Bag[190].Cat = 0) - DestCountSystem[30])

BufferClear[1] 		= ((D[6]> 0) AND (Line[31].SpaceBIT > 0) )
;BufferClear[2]		= ((Bag[Line[22].LastBag].Cat = 0) AND  (Line[22].SpaceBIT >= 1)); Empty bag buffer before CDC2
;BufferClear[3]		= ((Bag[Line[23].LastBag].Cat = 0) AND  (Line[23].SpaceBIT >= 1))
;BufferClear[4]		= (Bag[BufferBag[4]].Cat = 0) AND (RecircSpaces > 0) ;Recirc Valid
;BufferClear[5]		= ((Bag[BufferBag[5]].Cat = 0) AND (D[10] > 0) AND Request.DC[5] AND (Line[25].SpaceBIT >= 1))
;;BufferClear[6]		= (D[9] > 0) AND (Bag[BufferBag[6]].Cat = 0)
;BufferClear[7]		= (D[10] > 0) AND (Bag[BufferBag[7]].Cat = 0)

Uld[1].SDCReady 	= BufferClear[1]
Uld[2].SDCReady 	= FALSE
Uld[3].SDCReady		= FALSE
Uld[4].SDCReady 	= FALSE
;Uld[5].SDCReady 	= BufferClear[5]

Alarm[mySeq].Name 		= 0
Alarm[mySeq].Bag		= TransitBag
Alarm[mySeq].Beacon		= TRUE
Alarm[mySeq].Extra		= 0
Alarm[mySeq].Time		= 45000

;Setup Sequence
;--------------
STEP = D[900 + mySeq]
;Setup Pulse contact
PLS = (STEP <> LASTSTEP)
LASTSTEP = STEP

;Sequence Steps
;--------------
IF (STEP = 0) THEN
	;Disabled
ENDIF

;Step 1 - Reset Points
TON_10ms((STEP = 1),300,ResetPoints,ResetPointsET)
IF (STEP = 1) THEN
	O_Reset 	= TRUE
	FoundLine 	= 0
	Destination = 0
	IF (ResetPoints AND OffGoingEnable) THEN
		D[900+mySeq] = 2
	ENDIF
ENDIF

;Bags on storage line timers
R_TRIG(Std.Clock100ms,IncSettle)
AlarmBagNotProx 	= FALSE
AlarmBagNotProxLine = 0

LOOP n = MinLine TO MaxLine DO

	LineSettle[n]  = (I_BagAtStop[n] AND (Bag[Line[n].FirstBag].Cat > 0))
	IF IncSettle AND LineSettle[n] AND (BagSettledTime[n] < $FFFF) THEN
		BagSettledTime[n] = BagSettledTime[n] + 1
	ELSE IF NOT LineSettle[n] THEN
		BagSettledTime[n] = 0
		;If Bag has destiantion and not at stop then alarm
		IF (Bag[Line[n].FirstBag].Dst > 0) THEN
			Alarm[mySeq].Name	= almBagNotAtProx
			Alarm[mySeq].Bag	= Line[n].FirstBag
			Alarm[mySeq].Extra 	= n
		ENDIF
	ENDIF
		LongestSTime = 0
		LongestTime[n] = 0
ENDLOOP

LOOP n = MinLine TO MaxLine DO
	LineInList[n]  = FALSE
ENDLOOP

LOOP n = MinLine TO MaxLine DO
	LongestLine = 0
	LongestSTime = 0
	LOOP x = MinLine TO MaxLine DO
		IF (BagSettledTime[x] > LongestSTime) AND NOT LineInList[x] THEN ;(BagSettledTime[x] > BagSettledTime[n]) AND
			LongestSTime = BagSettledTime[x]
			LongestLine = x
		ENDIF
	ENDLOOP
	LineInList[LongestLine] = TRUE
	LongestTime[n] = LongestLine
ENDLOOP

;Buffer trip not correct alarms
LOOP n = 1 TO MaxBuffers DO
	IF (STEP = 2) AND BufferClear[n] AND NOT Uld[n].SDCReady THEN
		;Alarm[mySeq].Name 	= almSwitchFault - Not direct to buffers
		;Alarm[mySeq].Bag	= BufferBag[n]
	ENDIF
ENDLOOP

;Search for the bag with a valid destination that has been waiting the longest
IF STEP = 2 THEN

	FoundLine 	= 0
	Destination = 0
	BestTime 	= 0
	SettleTime = 30 ;3 seconds

	LOOP n = MinLine TO MaxLine DO
		IF ((BagSettledTime[n] > SettleTime) AND (BagSettledTime[n] > BestTime)) THEN
			SearchDest = Bag[Line[n].FirstBag].Dst

			SDC1_Valid  = (SearchDest = 31) AND Uld[1].SDCReady
			SDC2_Valid 	= (SearchDest = 32) AND Uld[2].SDCReady
			SDC3_Valid 	= (SearchDest = 33) AND Uld[3].SDCReady
			SDC4_Valid 	= (SearchDest = 34) AND Uld[4].SDCReady
;			SDC5_Valid 	= ((SearchDest = 35) AND Uld[5].SDCReady)
            ;SDC6_Valid 	= ((SearchDest = 36) AND Uld[6].SDCReady)
			;SDC7_Valid 	= ((SearchDest = 37) AND Uld[7].SDCReady)
			;RecircValid = ((SearchDest = 30) AND Line[20].Clear AND (Bag[Line[20].LastBag].Cat = 0))
			IF SDC1_Valid THEN
				FoundLine 	= n
				Destination = SearchDest
				BestTime 	= BagSettledTime[n]
			ENDIF
		ENDIF
	ENDLOOP

	IF ((FoundLine > 0) AND (Destination > 0) AND OffGoingEnable AND (Bag[TransitBag].Cat = 0)) THEN
		IF Line[myRelLine].Clear AND (Bag[Line[myRelLine].LastBag].Cat = 0) AND (Bag[TransitBag] .Cat = 0) AND NOT I_SDCBagAtBuffer[1] AND NOT O_SDCBufferOpen[1] THEN
			C[myRelLine] = 0
			D[900 + mySeq] = 3
		ENDIF
	ENDIF
ENDIF

;Step 3 - Select Line / Open Stop, Until Bag at correct destination
;Clear Line Selections
LOOP n = MinLine TO MaxLine DO
	LineSelect[n] = FALSE
ENDLOOP

IF (STEP = 3) THEN
	LineSelect[FoundLine] = TRUE
	IF (Destination >= 21) AND (Destination <= 21) THEN
		Uld[Destination - 20].DischargerStartLine = FoundLine ;Unloading Program
	ENDIF
	IF (Bag[TransitBag] .Cat = 0) AND (Bag[Line[FoundLine].FirstBag].Cat > 0)THEN
		IF PLS THEN
			Bag[TransitBag]  = Bag[Line[FoundLine].FirstBag]
			Bag[Line[FoundLine].FirstBag] 	= Bag[0]
		ENDIF
	ENDIF
	IF Line[myRelLine].Trip THEN
		Bag[Line[myRelLine].LastBag] = Bag[TransitBag]
		Bag[TransitBag] = Bag[0]
		D[900 + mySeq] = 1
	ENDIF
	Alarm[mySeq].Name	= almBagNotReleased
ENDIF

;Alarms
TimerAlarm.IN = NOT PLS AND (Alarm[mySeq].Name > 0)
TimerAlarm.PT = Alarm[mySeq].Time
TimerAlarm FUB TON_10ms()
Alarm[mySeq].On = TimerAlarm.Q
Alarm[mySeq].ET = TimerAlarm.ET

;Outputs
;-------

Y[71].Y07 = O_Reset
Y[71].Y08 = O_Reset
Y[72].Y07 = O_Reset
Y[72].Y08 = O_Reset
Y[73].Y07 = O_Reset
Y[73].Y08 = O_Reset
Y[74].Y07 = O_Reset
Y[74].Y08 = O_Reset
Y[75].Y07 = O_Reset
Y[75].Y08 = O_Reset

Y[71].Y05 = LineSelect[1]
Y[71].Y06 = LineSelect[2] OR LineSelect[1]
Y[71].Y03 = LineSelect[2]
Y[72].Y05 = LineSelect[3]
Y[72].Y06 = LineSelect[4]
Y[73].Y05 = LineSelect[5]
Y[73].Y06 = LineSelect[6]
Y[74].Y05 = LineSelect[7]
Y[74].Y06 = LineSelect[8]
Y[75].Y05 = LineSelect[9]
Y[75].Y06 = LineSelect[10]

END_PROGRAM
```

### Program Logical/BaseStandards/On_Offgoing/12_PN2 (IEC) - *Ongoing Sequence

#### x_pn.var
```iecst
VAR
	AlarmOld : UINT;
	Area : UINT;
	AreaChoice : ARRAY[0..4] OF UINT;
	AreaEndLine : UINT;
	AreaStartLine : UINT;
	AreaValid : BOOL;
END_VAR
VAR RETAIN
	Buff : UINT;
END_VAR
VAR
	Buffer : UINT;
	BufferBag : UINT;
	BufferBagNum : ARRAY[0..4] OF UINT;
	BufferCat : UDINT;
	BufferCus : UDINT;
	BufferDst : UINT;
	BufferPrg : UINT;
	BufferSettled : BOOL;
END_VAR
VAR RETAIN
	Dest : UINT;
END_VAR
VAR
	FoundDepth : UINT;
	I_BagatBuffer : ARRAY[0..4] OF BOOL;
END_VAR
VAR RETAIN
	LASTSTEP : UINT;
	LineSelect : ARRAY[0..19] OF BOOL;
END_VAR
VAR
	MaxBuffers : UINT;
	MaxDepth : UINT;
	MaxLine : UINT;
	MinLine : UINT;
	myDepth : UINT;
	myFound : UINT;
	myLine : UINT;
	myLineUsed : BOOL;
	myLineValid : BOOL;
	mySpace : UINT;
	n : UINT;
	O_OpenSelect : ARRAY[0..4] OF BOOL;
	O_Reset : BOOL;
	OnGoingEnable : BOOL;
END_VAR
VAR RETAIN
	PLS : BOOL;
END_VAR
VAR
	ResetPoints : BOOL;
	ResetPointsET : TIME;
	SearchBag : UINT;
	SettledBuffer : ARRAY[0..4] OF BOOL;
	SettledBufferET : ARRAY[0..4] OF TIME;
END_VAR
VAR RETAIN
	STEP : UINT;
END_VAR
VAR
	TestBuffer : UINT;
	TimerAlarm : TON_10ms;
	I_BagBagReleased : BOOL;
	mySeq : UINT;
	myZone : UINT;
	myTransitBag : UINT;
	myStartStop : UINT;
	O_OpenBuffer : ARRAY[0..9] OF BOOL;
END_VAR
```

#### x_pn.ab
```automation-basic
PROGRAM _CYCLIC

;--------------------------------------
;Sequence 4 - Ongoing To Storage D[900 + mySeq]
;--------------------------------------

;--------------------------------------------------------------------------------
;Revision 1.00 06/11/2009 D.J. First Issue - Automatic Line Allocation with Areas
;--------------------------------------------------------------------------------
mySeq 			= 4
myZone 			= 0
myTransitBag	= 298
myStartStop		= 100

IF (myStartStop >= 100) THEN
	myStartStop = myStartStop + 7600
ENDIF

;Inputs
OnGoingEnable 		= ((D[mySeq] > 0) AND NOT Std.HaltSysZone[myZone])

I_BagatBuffer[1]		= Request.VC[2]
I_BagatBuffer[2]		= FALSE
I_BagatBuffer[3]		= FALSE
I_BagatBuffer[4]		= FALSE

O_Reset 		  		= FALSE
O_OpenSelect[1]			= FALSE
O_OpenSelect[2]			= FALSE
O_OpenSelect[3]			= FALSE
O_OpenSelect[4]			= FALSE

O_OpenBuffer[1]			= FALSE
O_OpenBuffer[2]			= FALSE
O_OpenBuffer[3]			= FALSE
O_OpenBuffer[4]			= FALSE

MaxBuffers 			= 1 	;Set Max Buffers to search
MinLine				= 6 	;Set First Storage Line
MaxLine				= 11		;Set Last Storage Line
MaxDepth			= 9    ;Capacity of the longest line - used in search

Alarm[mySeq].Name 		= 0
Alarm[mySeq].Bag		= myTransitBag
Alarm[mySeq].Beacon		= TRUE
Alarm[mySeq].Extra	 	= 0
Alarm[mySeq].Time		= 6000

;Setup Sequence
;--------------
STEP = D[900 + mySeq]
;Setup Pulse contact
PLS = (STEP <> LASTSTEP)
LASTSTEP = STEP

;Step 0 - Disabled
IF (STEP = 0) THEN
	;Disabled
ENDIF

;Step 1 - Reset Ongoing Points
TON_10ms((STEP = 1),300,ResetPoints,ResetPointsET)
IF (STEP = 1) THEN
	Dest  	= 0
	Buff 	= 0
	O_Reset = TRUE
	IF (ResetPoints AND OnGoingEnable) THEN
		D[900 + mySeq] = 2
	ENDIF
ENDIF

;Bag Settles at each buffer
TON_10ms(I_BagatBuffer[1],300,SettledBuffer[1],SettledBufferET[1])
;TON_10ms(I_BagatBuffer[2],300,SettledBuffer[2],SettledBufferET[2])
;TON_10ms(I_BagatBuffer[3],300,SettledBuffer[3],SettledBufferET[3])

BufferBagNum[1]	    = 296
;BufferBagNum[2]	= 161
;BufferBagNum[3]	= myTransitBag

;Step 2 - Search for a valid Bag at one of the buffers
IF (STEP = 2) THEN

	Buff 	= 0
	Dest 	= 0

	IF OnGoingEnable THEN

		Alarm[mySeq].Name 	= almNoAlarm

		;Search only 1 buffer bag per scan/task
		Buffer = Buffer + 1
		IF Buffer > MaxBuffers THEN
			Buffer = 1
		ENDIF
		;Set Test Value for Monitoring
		IF TestBuffer > 0 THEN
			Buffer = TestBuffer
		ENDIF

		BufferBag		= BufferBagNum[Buffer]
		BufferSettled 	= SettledBuffer[Buffer]
		BufferPrg 		= Bag[BufferBag].Prg
		BufferCat		= Bag[BufferBag].Cat
		BufferCus		= Bag[BufferBag].Cus
		BufferDst 		= Bag[BufferBag].Dst

		IF (BufferSettled AND (BufferCat > 0) AND (BufferPrg > 0) AND (BufferPrg <= Std.MaxProg) AND (OnGoingEnable)) THEN

			;Manual Destination has been set?
			IF (BufferDst > 0) THEN

				n = BufferDst
				IF ((n >= MinLine) AND (n <= MaxLine) AND (Line[n].Space > 0) AND Line[n].Clear) THEN
					Dest 	= n
					Buff 	= Buffer
					D[900 + mySeq] 	= 3
				ELSE
					Alarm[mySeq].Name 	= almDestinationNotValid
					Alarm[mySeq].Bag	= BufferBag
				ENDIF

			ELSE IF Std.AutoLineAllocation THEN ;/BufferDst > 0

				;Search Each Storage Area
				AreaChoice[1] = D[3000 + BufferPrg]
				AreaChoice[2] = D[3100 + BufferPrg]
				AreaChoice[3] = D[3200 + BufferPrg]
				AreaChoice[4] = D[3300 + BufferPrg]

				LOOP Area = 1 TO 4 DO

					AreaStartLine 	= D[250 + AreaChoice[Area]]
					AreaEndLine 	= D[270 + AreaChoice[Area]]
					AreaValid		= ((AreaStartLine > 0) AND (AreaEndLine > 0) AND (AreaEndLine >= AreaStartLine))
					IF AreaValid THEN

						;Search for a line with the same program
						;---------------------------------------
						LOOP myLine = AreaStartLine TO AreaEndLine DO
							myLineValid = ((myLine >= MinLine) AND (myLine <= MaxLine))
							myLineUsed	= (D[myStartStop + myLine] > 0) ;Start / Stop On
							IF myLineValid AND myLineUsed THEN
								n 			= myLine
								SearchBag 	= (Line[n].LastBag - Line[n].Space)
								IF ((SearchBag >= Line[n].FirstBag) AND (Bag[SearchBag].Prg = BufferPrg) AND (Line[n].Space > 0) AND Line[n].Clear) THEN
									;Found line with a matching program
									Dest 	= n
								ENDIF ;/SearchBag
							ENDIF ;/myLineValid
							EXITIF (Dest <> 0)
						ENDLOOP ;/myLine loop

						;Search for an empty line
						;------------------------
						IF (Dest = 0) THEN
							LOOP myLine = AreaStartLine TO AreaEndLine DO
								myLineValid = ((myLine >= MinLine) AND (myLine <= MaxLine))
								myLineUsed	= (D[myStartStop + myLine] > 0) ;Start / Stop On
								IF myLineValid AND myLineUsed THEN
									n 			= myLine
									SearchBag 	= (Line[n].FirstBag)
									IF ((Bag[SearchBag].Prg = 0) AND (Line[n].Space > 0) AND Line[n].Clear) THEN
										;Found line with a matching program
										Dest 	= n
									ENDIF ;/SearchBag
								ENDIF ;/myLineValid
							EXITIF (Dest <> 0)
							ENDLOOP ;/myLine loop
						ENDIF ;/Dest = 0

						;Search for a line that already contains a bag with the same program starting at the back
						;----------------------------------------------------------------------------------------
						IF (Dest = 0) THEN
							LOOP myDepth = (MaxDepth - 2) DOWNTO 0 DO ;Don't search the last bag as the line would already be full!!
								LOOP myLine = AreaStartLine TO AreaEndLine DO
									myLineValid = ((myLine >= MinLine) AND (myLine <= MaxLine))
									myLineUsed	= (D[myStartStop + myLine] > 0) ;Start / Stop On
									IF myLineValid AND myLineUsed THEN
										n 			= myLine
										SearchBag 	= (Line[n].FirstBag + myDepth)
										IF ((Bag[SearchBag].Prg = BufferPrg) AND (Line[n].Space > 0) AND Line[n].Clear) THEN
											;Found line with a matching program
											FoundDepth 	= myDepth
											Dest 		= n
										ENDIF ;/SearchBag
									ENDIF ;/myLineValid
									EXITIF (Dest <> 0)
								ENDLOOP ;/myLine loop
								EXITIF (Dest <> 0)
							ENDLOOP ;/myDepgh
						ENDIF ;/Dest = 0

						;Search for line with the most space
						;-----------------------------------
						IF (Dest = 0) THEN
							mySpace = 0
							myFound	= 0
							LOOP myLine = AreaStartLine TO AreaEndLine DO
								myLineValid = ((myLine >= MinLine) AND (myLine <= MaxLine))
								myLineUsed	= (D[myStartStop + myLine] > 0) ;Start / Stop On
								IF myLineValid AND myLineUsed THEN
									n 			= myLine
									SearchBag 	= (Line[n].LastBag)
									IF ((Bag[SearchBag].Prg = 0) AND (Line[n].Space > mySpace) AND Line[n].Clear) THEN
										;Found line with a matching program
										myFound	= n
										mySpace = Line[n].Space
									ENDIF ;/SearchBag
								ENDIF ;/myLineValid
							ENDLOOP ;/myLine loop

							IF (myFound > 0) THEN
								Dest 	= myFound
							ENDIF

						ENDIF ;/Dest = 0

					ENDIF ;/Area Valid
					EXITIF (Dest <> 0)
				ENDLOOP ;/Area Loop

			ENDIF ;/BufferDst > 0

			;Destination line found!!
			IF (Dest <> 0) THEN
				Buff = Buffer
				IF (Bag[myTransitBag].Cat = 0) AND (Bag[BufferBagNum[Buff]].Cat > 0) THEN ;Bag in Transit
					Bag[BufferBagNum[Buff]].Dst = USINT(Dest)
					Bag[myTransitBag]	= Bag[BufferBagNum[Buff]]
					Bag[BufferBagNum[Buff]]	 	= Bag[0]
					C[Dest] = 0
					D[900 + mySeq] 	= 3 ; Open buffer
				ENDIF
			ELSE
				;Storage full!!
				;Do Nothing? Alarm?
				;Other Area?
			ENDIF

		ENDIF ;/BagSettled

		;Buffer Alarms
		IF (BufferPrg > 0) AND NOT BufferSettled THEN
			Alarm[mySeq].Name 	= almBagNotAtProx
			Alarm[mySeq].Bag	= BufferBag
		ELSE IF (BufferPrg = 0) AND BufferSettled THEN
			Alarm[mySeq].Name 	= almBagNotShownOnScreen
			Alarm[mySeq].Bag	= BufferBag
		ENDIF
	ENDIF
ENDIF

;Clear Line Selections
LOOP n = 1 TO Std.MaxLines DO
	LineSelect[n] = FALSE
ENDLOOP

;Step 3 - Select line / open buffer stop
IF (STEP = 3) THEN
	LineSelect[Dest] 	= TRUE
	O_OpenBuffer[Buff] = TRUE
	;Bag arrived on selected line
	IF Line[Dest].Trip THEN
		D32[498] 					= Bag[myTransitBag].Cus	;Set Customer for Customer FIFO
		Bag[myTransitBag].Dst 		= 0 		    ;Clear Destination
		Bag[Line[Dest].LastBag] 	= Bag[myTransitBag]
		Bag[myTransitBag] 			= Bag[0]
		D[900 + mySeq] 				= 1
	ENDIF
	Alarm[mySeq].Name = almBagNotArrived
ENDIF

;Alarms
TimerAlarm.IN = NOT PLS AND (Alarm[mySeq].Name > 0) AND (AlarmOld = Alarm[mySeq].Name)
TimerAlarm.PT = Alarm[mySeq].Time
TimerAlarm FUB TON_10ms()
Alarm[mySeq].On = TimerAlarm.Q
Alarm[mySeq].ET = TimerAlarm.ET

AlarmOld = Alarm[mySeq].Name ;Need to ensure alarm changes as may be multiple alarms on step 2

Enable.PN[1] = O_OpenBuffer[1]

;Outputs
Y[4].Y06 = LineSelect[6]

Y[4].Y07 = LineSelect[7]
Y[4].Y08 = LineSelect[8]
Y[4].Y09 = LineSelect[9]
Y[4].Y10 = LineSelect[10]
Y[4].Y11 = LineSelect[11]
Y[4].Y15 =  O_Reset

END_PROGRAM
```

### Program Logical/BaseStandards/On_Offgoing/13_spf2 (IEC, version 1.00.0) - * Soiled Offgoing Transfer Lines 1 - 14

#### 5_spf1Cyclic.ab
```automation-basic
PROGRAM _CYCLIC
	(* cyclic program *)

;----------------------------------------
;Sequence 5 - SPF1 Offgoing Points D[905]
;----------------------------------------
;Inputs
;------

OffGoingEnable 		= ((D[15] > 0) AND NOT Std.HaltSys)

I_BagAtStop[6] 		= X[5].X06 OR testAtStop;(Bag[Line[6].FirstBag].Cat > 0);X[5].X06
I_BagAtStop[7] 		= X[5].X07 OR testAtStop;(Bag[Line[7].FirstBag].Cat > 0);X[5].X07
I_BagAtStop[8] 		= X[5].X08 OR testAtStop;(Bag[Line[8].FirstBag].Cat > 0);X[5].X08
I_BagAtStop[9] 		= X[5].X09 OR testAtStop;(Bag[Line[9].FirstBag].Cat > 0);X[5].X09
I_BagAtStop[10] 	= X[5].X10 OR testAtStop;(Bag[Line[10].FirstBag].Cat > 0);X[5].X10
I_BagAtStop[11] 	= X[5].X11 OR testAtStop;(Bag[Line[11].FirstBag].Cat > 0);X[5].X11

O_Reset 			= FALSE

;Buffer line configuration
;-------------------------
MaxBuffers			= 2

BufferBag[1]		= 266;Last buffer bag number
BufferBag[2]		= 280 ;Last buffer bag number
	BufferBag[4]		= 246 ;Last buffer bag number

;Banbury Special - Empty bags from SDC2 travel on a rail close to Lines 6-14
;---------------------------------------------------------------------------

BufferClear[1] 		= ( (Line[21].SpaceBIT > 0) AND (Bag[269].Cat = 0) AND (D[21] > 0) AND (Bag[BufferBag[1]].Cat = 0))
BufferClear[2]		= ((Line[22].SpaceBIT > 0)  AND (D[22] > 0) AND (Bag[BufferBag[2]].Cat = 0))

;Alternating between SDC1 and SDC3

Uld[1].SDCReady 	= (BufferClear[1] ) ;Passed to unloading search
Uld[2].SDCReady 	= (BufferClear[2] );Passed to unloading search

Alarm[5].Name 		= 0
Alarm[5].Bag		= 324
Alarm[5].Beacon		= TRUE
Alarm[5].Extra		= 0
Alarm[5].Time		= 3000

;Setup Sequence
;--------------
STEP = D[905]
;Setup Pulse contact
PLS = (STEP <> LASTSTEP)
LASTSTEP = STEP

;Sequence Steps
;--------------
IF (STEP = 0) THEN
	;Disabled
ENDIF

;Step 1 - Reset Points
TON_10ms((STEP = 1),300,ResetPoints,ResetPointsET)
IF (STEP = 1) THEN
	O_Reset 	= TRUE
	FoundLine 	= 0
	Destination = 0
	;IF (ResetPoints AND OffGoingEnable) THEN
	IF (ResetPoints AND OffGoingEnable AND NOT I_BagReleased) THEN
		D[905] = 2
	ENDIF
ENDIF

;Bags on storage line timers
R_TRIG(Std.Clock100ms,IncSettle)
AlarmBagNotProx 	= FALSE
AlarmBagNotProxLine = 0

LOOP n = 1 TO Std.MaxLines DO

	LineSettle[n]  = (I_BagAtStop[n] AND (Bag[Line[n].FirstBag].Cat > 0))
	IF IncSettle AND LineSettle[n] AND (BagSettledTime[n] < $FFFF) THEN
		BagSettledTime[n] = BagSettledTime[n] + 1
	ELSE IF NOT LineSettle[n] THEN
		BagSettledTime[n] = 0
		;If Bag has destiantion and not at stop then alarm
		IF (STEP = 2) AND (Bag[Line[n].FirstBag].Dst > 0) THEN
			Alarm[5].Name	= almBagNotAtProx
			Alarm[5].Bag	= Line[n].FirstBag
			Alarm[5].Extra 	= n
		ENDIF
	ENDIF

ENDLOOP

;Buffer trip not correct alarms
LOOP n = 1 TO MaxBuffers DO
	IF (STEP = 2) AND BufferClear[n] AND NOT Uld[n].SDCReady THEN
		Alarm[5].Name 	= almSwitchFault
		Alarm[5].Bag	= BufferBag[n]
	ENDIF
ENDLOOP

;Search for the bag with a valid destination that has been waiting the longest
IF STEP = 2 THEN

	FoundLine 	= 0
	Destination = 0
	BestTime 	= 0
	SettleTime = 30 ;3 seconds

	LOOP n = 1 TO Std.MaxLines DO

		IF (BagSettledTime[n] > SettleTime) THEN
			SearchDest = Bag[Line[n].FirstBag].Dst

			SDC1_Valid  = ((SearchDest = 21) AND Uld[1].SDCReady AND (Line[21].SpaceBIT > 0))
			SDC2_Valid 	= ((SearchDest = 22) AND Uld[2].SDCReady AND (Line[22].SpaceBIT > 0))

			IF (SDC1_Valid OR SDC2_Valid ) THEN
				FoundLine 	= n
				Destination = SearchDest
				BestTime 	= BagSettledTime[n]
			ENDIF
		ENDIF

	ENDLOOP

	IF ((FoundLine > 0) AND OffGoingEnable AND (Bag[318].Cat = 0) AND Line[13].Clear AND (Bag[321].Cat = 0)) THEN
		D[905] = 3
	ENDIF

ENDIF

;Step 3 - Select Line / Open Stop, Until Bag at correct destination
;Clear Line Selections
LOOP n = 6 TO Std.MaxLines DO
	LineSelect[n] = FALSE
	Indication[n] = FALSE
ENDLOOP

IF (STEP = 3) THEN

	IF PLS THEN
		C[13] = 0
	ENDIF

	IF PLS  AND (Bag[318].Cat = 0) AND (Bag[Line[FoundLine].FirstBag].Cat > 0)THEN
		Bag[318] 						= Bag[Line[FoundLine].FirstBag]
		Bag[Line[FoundLine].FirstBag] 	= Bag[0]
	ENDIF

	;Select Line - Wait for bag to arrive
	LineSelect[FoundLine] = TRUE ;TRUE
	Indication[FoundLine] = TRUE ;Use indication as single stop and display dosen't indicate to operator where the bag is comming from

	;Select Route
	IF (Destination = 21) OR (Destination = 22) THEN
		Uld[1].DischargerStartLine = FoundLine ;Unloading Program

		IF ((C[13] > 0) AND NOT PLS) THEN
			IF ((Bag[318].Cat > 0) AND (Bag[321].Cat = 0))THEN

				Bag[321] 	= Bag[318]
				Bag[318] 	= Bag[0]
				D[905] 		= 1
			ENDIF
		ENDIF

ENDIF

	Alarm[5].Name	= almBagNotReleased

ELSE

ENDIF

;SSR2 Brush speed reducer

;Alarms
TimerAlarm.IN = NOT PLS AND (Alarm[5].Name > 0)
TimerAlarm.PT = Alarm[5].Time
TimerAlarm FUB TON_10ms()
Alarm[5].On = TimerAlarm.Q
Alarm[5].ET = TimerAlarm.ET

;Outputs
;-------
Y[5].Y15 = O_Reset

Y[5].Y06 = LineSelect[6]
Y[5].Y07 = LineSelect[7]
Y[5].Y08 = LineSelect[8]
Y[5].Y09 = LineSelect[9]
Y[5].Y10 = LineSelect[10]
Y[5].Y11 = LineSelect[11]

END_PROGRAM
```

### Program Logical/BaseStandards/On_Offgoing/14_svc4 (IEC) - * SVC3 Vertical Conveyor

#### 18_svc3.var
```iecst
VAR RETAIN
	STEP : UINT;
	PLS : BOOL;
	LASTSTEP : UINT;
	O_OpenBufferStop : BOOL;
	I_BagAtBuffer : BOOL;
	O_RunMotor : BOOL;
	BagSettled : BOOL;
	BagSettledET : TIME;
	BagAtBuffer : BOOL;
	RunOnET : TIME;
	RunOn : BOOL;
	BagNearTopET : TIME;
	BagNearTop : BOOL;
	BagAtBufferET : UDINT;
	I_BagInIncline : BOOL;
END_VAR
VAR
	I_BagAtOutgoingBuffer : BOOL;
	zzTON_10ms00002 : TON_10ms;
	zzTON_10ms00003 : TON_10ms;
	I_PaddleInPosition : BOOL;
	zzTON_10ms00004 : TON_10ms;
	CloseBufferStop : BOOL;
	CloseBufferStopET : TIME;
	O_OutgoingBufferOpen : BOOL;
	TimerAlarm : TON_10ms;
	O_SelectSP4ToSP2 : BOOL;
	I_BagReleased : BOOL;
	O_SelectSP4 : BOOL;
	I_BagOutAtTop : BOOL;
	I_BagOutAtBottom : BOOL;
	I_BagOnCarriage : BOOL;
	I_CarriageAtTop : BOOL;
	I_CarriageAtBottom : BOOL;
	O_OpenCarriageStop : BOOL;
	O_MoveUp : BOOL;
	O_MoveDown : BOOL;
	I_BagAtBufferStop : BOOL;
	BagSettledAtBuffer : BOOL;
	BagSettledAtBufferET : TIME;
	BufferClear : BOOL;
	I_BagOutAtTopSVC3 : BOOL;
	I_CarrAtTop : BOOL;
	I_CarrAtBottom : BOOL;
	I_CarrAtFullBagIn : BOOL;
	I_BagOnCarr : BOOL;
	O_SP1Bend : BOOL;
	O_SP3Straight : BOOL;
	O_SP8Bend : BOOL;
	O_OpenBuffer : BOOL;
	O_MoveCarrUp : BOOL;
	O_MoveCarrDown : BOOL;
	O_OpenCarrStop : BOOL;
	O_SP3Bend : BOOL;
	SettledBuffer : BOOL;
	SettledBufferET : UDINT;
	ParingLoopEnabled : BOOL;
	BagSettledOnCarr : BOOL;
	BagSettledOnCarrET : UDINT;
	PairOnLoop : BOOL;
	PairNotValidSVC3 : BOOL;
	HLBagMatch : BOOL;
	NoPairForSVC3 : BOOL;
	LLBagMatch : BOOL;
	CarriagePasted : BOOL;
	CarriagePastedET : UDINT;
END_VAR
```

#### 18_svc3Cyclic.ab
```automation-basic
PROGRAM _CYCLIC
	(* cyclic program *)

;---------------------------------------------------
;Sequence 13 - SIC2 Soiled Incline Conveyor 2 D[913]
;---------------------------------------------------

;Inputs
I_CarrAtTop				= X[10].X08
I_CarrAtBottom			= X[10].X09
I_CarrAtFullBagIn       = X[10].X10
I_BagOnCarr				= X[10].X11

I_BagReleased			= X[10].X13
I_BagAtBuffer			= X[10].X12

O_SP1Bend   			= FALSE ;Y301
O_SP3Straight			= FALSE ;Y311
O_SP8Bend               = FALSE ;Y314

O_OpenBuffer			= FALSE
O_MoveCarrUp			= FALSE
O_MoveCarrDown			= FALSE
O_OpenCarrStop			= FALSE
O_SP3Bend               = FALSE

Request.SVC1LowLevel    = FALSE
Request.SVC3LowLevel    = FALSE

Alarm[10].Name 			= 0
Alarm[10].Bag			= 310
Alarm[10].Beacon		= TRUE
Alarm[10].Extra			= 0
Alarm[10].Time			= 3000
;Setup Sequence
STEP = D[910]
;Setup Pulse contact
PLS = (STEP <> LASTSTEP)
LASTSTEP = STEP

;Sequence
;Step 0 - Disabled
IF (STEP = 0) THEN
	;Disabled
ENDIF

;Move carriage down to top full bag in
IF (STEP = 1) THEN
	O_MoveCarrDown = NOT I_CarrAtFullBagIn
	IF I_CarrAtFullBagIn THEN
		D[910] = 2
	ENDIF
	IF NOT Std.EStop THEN
		Alarm[10].Name = almCarriageMoveFault
	ENDIF
ENDIF

;check status
IF (STEP = 2) THEN
	IF (NOT I_BagOnCarr AND NOT I_CarrAtBottom AND NOT I_CarrAtTop) THEN
		D[910] = 3
	ENDIF
	IF I_BagOnCarr OR I_CarrAtBottom OR I_CarrAtTop THEN
		Alarm[10].Name = almSwitchFault
	ENDIF
ENDIF

;Bag at Pairing loop buffer stop
TON_10ms(I_BagAtBuffer,300,SettledBuffer,SettledBufferET)
IF (STEP = 3) THEN
	IF SettledBuffer AND NOT Std.HaltSys AND ParingLoopEnabled THEN
		D[910] = 4
	ENDIF
ENDIF

;Open Buffer stop - Enable
IF (STEP = 4) THEN
	O_OpenBuffer 	= (NOT I_BagOnCarr AND I_CarrAtFullBagIn)

	IF I_BagOnCarr THEN
		IF ((Bag[305].Cat > 0) AND (Bag[310].Cat = 0)) THEN
			Bag[310] = Bag[305]
			Bag[305] = Bag[0]
		ENDIF
		D[910] = 5
	ENDIF
	Alarm[10].Name = almBagNotArrived
ENDIF

;Let bag settle on carriage and decide where bag is going
TON_10ms(I_BagOnCarr,300,BagSettledOnCarr,BagSettledOnCarrET)
IF (STEP = 5) THEN

	IF (BagSettledOnCarr AND (Bag[310].Cat > 0)	AND ParingLoopEnabled) THEN

		;IF ((LoopPair = 1) AND (LoopPairDest = Bag[310].Dst)) THEN
		IF (PairOnLoop AND (Bag[310].Cnt = 1)) THEN
			IF ((Bag[310].Dst >= 6) AND (Bag[310].Dst <= 12)) THEN
				D[910] = 6 ;check that loop pair is not being split up by single bag on loop with dest
			ELSE IF ((Bag[310].Dst >= 0) AND (Bag[310].Dst <= 5)) THEN
				D[910] = 11
			ENDIF
			ELSE
			D[910] = 6
		ENDIF

		IF ((Bag[310].Dst = 0) OR PairNotValidSVC3) THEN
			D[910] = 6 	;Not correct bag then recirc
		ELSE IF ((Bag[310].Dst >= 6) AND (Bag[310].Dst <= 12)AND NOT PairOnLoop)  THEN
			D[910] = 6 	;Bag for high-level storage
		ELSE IF ((Bag[310].Dst > 0) AND (Bag[310].Dst <=5) AND NOT PairOnLoop)  THEN
			D[910] = 11 ;Bag for low-level storage
		ENDIF
	ENDIF

	IF NOT I_BagOnCarr THEN
		Alarm[10].Name = almBagNotSettled
	ENDIF
ENDIF

;Move Carriage Up to top position
IF (STEP = 6) THEN
	O_MoveCarrUp = NOT I_CarrAtTop
	IF I_CarrAtTop THEN
		D[910] = 7
	ENDIF
	IF NOT Std.EStop THEN
		Alarm[10].Name = almCarriageMoveFault
	ENDIF
ENDIF

;Request to SPN 1 if bag has destination
;recirculate if bag has no dest and space on H/L buffer
IF (STEP = 7) THEN

	IF (PairOnLoop AND (Bag[310].Cnt = 0) AND (Bag[304].Cat = 0)) THEN
		IF Line[17].Clear THEN
			D[910] = 8
		ENDIF
	ELSE

	IF ((Bag[310].Cat = Bag[296].Cat) AND (Bag[310].Dst = Bag[296].Dst)) THEN
		HLBagMatch = TRUE ;SVC2 bag is the pair then set request release
	ELSE IF NoPairForSVC3 THEN
		HLBagMatch = TRUE ;SVC3 Bag has no pair in transit then set request release
	ELSE
		HLBagMatch = FALSE
	ENDIF

	;Sometimes the bag is paired whilst on SVC3 carriage and needs to be sent to the low-level
	IF ((Bag[310].Cat > 0) AND (Bag[310].Dst > 0) AND (Bag[310].Dst <=5))  THEN
			D[910] = 11 ;Bag for low-level storage
	ELSE IF (HLBagMatch AND (Bag[310].Dst > 5) AND (Bag[310].Dst < 12))  THEN
	 	Request.SVC3HighLevel = I_CarrAtTop
	ENDIF
	ENDIF

	IF Enable.SVC3HighLevel THEN
		D[910] = 9
	ELSE IF (((Bag[310].Dst = 0) OR PairNotValidSVC3) AND (Bag[304].Cat = 0) AND Line[17].Clear) THEN
		D[910] = 8
	ENDIF

ELSE
	Request.SVC3HighLevel = FALSE
ENDIF

;send bag back onto pairing loop
IF (STEP = 8) THEN
	O_OpenCarrStop = I_CarrAtTop
	O_SP3Bend      = TRUE
	IF PLS THEN
		C[17] = 0
	ENDIF
	IF Line[17].Trip THEN
		IF((Bag[310].Cat > 0) AND (Bag[304].Cat = 0)) THEN
			Bag[304] = Bag[310]
			Bag[310] = Bag[0]
		ENDIF
		D[910] = 10
	ENDIF
	IF NOT Std.EStop THEN
		Alarm[10].Name = almBagNotReleased
	ENDIF
ENDIF

;Open carriage stop and move to ongoing
IF (STEP = 9) THEN
	O_OpenCarrStop = I_CarrAtTop
	O_SP3Straight  = TRUE
	O_SP1Bend      = TRUE
	IF I_BagReleased THEN
		D[910] = 10
	ENDIF

	IF NOT Std.EStop THEN
		Alarm[10].Name = almBagNotReleased
	ENDIF
ENDIF

;Check roller  switch
IF (STEP = 10) THEN
	IF NOT I_CarrAtFullBagIn AND NOT I_BagOnCarr THEN
		D[910] = 1
	ENDIF
	Alarm[10].Name = almSwitchFault
ENDIF

;Check roller  switch
IF (STEP = 11) THEN
	IF NOT I_CarrAtBottom  THEN
		D[910] = 12
	ENDIF
	Alarm[10].Name = almSwitchFault
ENDIF

;send bag down to low level
IF (STEP = 12) THEN
	O_MoveCarrDown = NOT I_CarrAtBottom
	IF I_CarrAtBottom AND NOT Enable.SVC1LowLevel  THEN
		D[910] = 13
	ENDIF
ENDIF

;request low level ongoing
IF (STEP = 13) THEN

	IF ((Bag[310].Cat = Bag[296].Cat) AND (Bag[310].Dst = Bag[296].Dst)) THEN
		LLBagMatch = TRUE ;SVC2 bag is the pair then set request release
	ELSE IF NoPairForSVC3 THEN
		LLBagMatch = TRUE ;SVC3 Bag has no pair in transit then set request release
	ELSE
		LLBagMatch = FALSE
	ENDIF

	IF (LLBagMatch AND (Bag[310].Dst > 0) AND (Bag[310].Dst <= 5))  THEN
	 	Request.SVC3LowLevel = I_CarrAtBottom
	ENDIF

	IF Enable.SVC3LowLevel THEN
		D[910] = 14
	ENDIF
ENDIF

;open carriage stop
IF (STEP = 14) THEN
	O_OpenCarrStop = I_CarrAtBottom
	O_SP8Bend      = TRUE
	IF PLS THEN
		C[28] = 0
	ENDIF
	IF (C[28] > 1) THEN
		D[910] = 15
	ENDIF
ENDIF

;Check switches
IF (STEP = 15) THEN
	IF NOT I_CarrAtTop AND NOT I_CarrAtFullBagIn AND NOT I_BagOnCarr THEN
		D[910] = 16
	ENDIF
	IF NOT Std.EStop THEN
		Alarm[10].Name = almSwitchFault
	ENDIF
ENDIF

;move up passed full bag in
IF STEP = 16 THEN
	O_MoveCarrUp = NOT I_CarrAtTop
	IF I_CarrAtFullBagIn THEN
		D[910] = 17
	ENDIF
ENDIF

;carriage is pasted full bag in
TON_10ms(NOT I_CarrAtFullBagIn,30,CarriagePasted,CarriagePastedET)
IF (STEP = 17) THEN
	O_MoveCarrUp = NOT I_CarrAtTop
	IF CarriagePasted THEN
		D[910] = 1
	ENDIF
ENDIF

;Alarms
TimerAlarm.IN 	= NOT PLS AND (Alarm[10].Name > 0)
TimerAlarm.PT 	= Alarm[10].Time
TimerAlarm FUB TON_10ms()
Alarm[10].On 	= TimerAlarm.Q
Alarm[10].ET 	= TimerAlarm.ET

;PLC Outputs
;-----------
Y[3].Y11        = O_SP3Straight
Y[3].Y10        = O_SP3Bend
Y[3].Y01        = O_SP1Bend
Y[3].Y14        = O_SP8Bend
Y[10].Y12 		= O_OpenBuffer
Y[12].Y09 		= (O_MoveCarrUp 	AND NOT I_CarrAtTop)
Y[12].Y10 		= O_MoveCarrDown

Y[12].Y12 		= O_OpenCarrStop

;Don't allow forcing of carriage movement and carriage stop
YForceDisable[12].Y09 = TRUE
YForceDisable[12].Y06 = TRUE
YForceDisable[12].Y07 = TRUE
YForceDisable[12].Y12 = TRUE

END_PROGRAM
```

### Package Logical/BaseStandards/Points - Standard Points

- Standard Sequence 1_x_Point V2.00.2 ENG.docx (binary file, 205347 bytes)
- Standard Sequence x_1_Point V2.00.4 ENG.docx (binary file, 206472 bytes)
### Program Logical/BaseStandards/Points/ComplexPoints/1_x_Point (IEC, version 2.00.3) - *Point control for 1 line into x buffers

#### 1_x_Point.var - Local variables
```iecst
(********************************************************************
 * COPYRIGHT -- HP
 ********************************************************************
 * Program: 1_x_Point
 * File: 1_x_Point.var
 * Author: treamsbottom
 * Created: March 13, 2015
 ********************************************************************
 * Local variables of program 1_x_Point
 ********************************************************************)
VAR CONSTANT
	LOCAL_MAX_DESTS : UINT := 2;
END_VAR
VAR
	mySeq : UINT;
	no_RecieveLines : UINT;
	myRelLine : ARRAY[0..LOCAL_MAX_DESTS] OF UINT;
	useDestinations : BOOL;
	myRelLineDest : ARRAY[0..LOCAL_MAX_DESTS] OF relLineDest_typ;
	myZone : UINT;
	myIO : UINT;
	myBag : UINT;
	i_bagAtBuffer : BOOL;
	x : UINT;
	i_bagAtBufferOut : ARRAY[0..LOCAL_MAX_DESTS] OF BOOL;
	i_bufferOutOpen : ARRAY[0..LOCAL_MAX_DESTS] OF BOOL;
	n : UINT;
	bufferClear : ARRAY[0..LOCAL_MAX_DESTS] OF BOOL;
	myOutBag : ARRAY[0..LOCAL_MAX_DESTS] OF UINT;
	o_select : ARRAY[0..LOCAL_MAX_DESTS] OF BOOL;
	o_reset : BOOL;
	o_openBuffer : BOOL;
	step : UINT;
	pls : BOOL;
	lastStep : UINT;
	alt : UINT;
	myLine : UINT;
	releaseValid : BOOL;
	ton_10ms_reset : TON_10ms;
	ton_10ms_SettledBuffer : TON_10ms;
	timerAlarm : TON_10ms;
	bagArrived : ARRAY[0..LOCAL_MAX_DESTS] OF BOOL;
	bagReleased : BOOL;
	myTransitBag : UINT;
	bufferSettleTime : UDINT;
	myPoint : UINT;
END_VAR
```

#### 1_x_Point.typ - Local data types
```iecst
(********************************************************************
 * COPYRIGHT -- HP
 ********************************************************************
 * Program: 1_x_Point
 * File: 1_x_Point.typ
 * Author: treamsbottom
 * Created: March 13, 2015
 ********************************************************************
 * Local data types of program 1_x_Point
 ********************************************************************)

TYPE
	relLineDest_typ : 	STRUCT
		dest : ARRAY[0..LOCAL_MAX_DESTS]OF UINT;
	END_STRUCT;
END_TYPE
```

#### 1_x_Point.st - Implementation code
```iecst
(********************************************************************
* COPYRIGHT -- HP
********************************************************************
* PROGRAM: 1_x_Point
* File: 1_x_Point.st
* Author: treamsbottom
* Created: March 13, 2015
********************************************************************
* Implementation OF PROGRAM 1_x_Point
********************************************************************)
//Version 1.0.0 First Release.
//Version 1.01.0 - Split buffer clear and bag arrive vars..
//Version 2.00.1 - Add transit bag position to comply with new Standards. First release with new standards.
//Version 2.00.2 - Make transit bag optional..
PROGRAM _INIT
//Configuration
mySeq						:= 13;	//Sequence number
no_RecieveLines				:= LOCAL_MAX_DESTS;	//Number of lines buffer can send to.
myPoint						:= 6;

myRelLine[1]				:= 0;
myRelLine[2]				:= 0;

useDestinations 			:= 0; 		// Use bag dest to route bag
myRelLineDest[1].dest[1]	:= 32; 	// Destination in bag if different to buffer...
myRelLineDest[1].dest[2]	:= 33;

myRelLineDest[2].dest[1]	:= 31;

myZone						:= 1;
myIO						:= 106;
myBag						:= 0; //Buffer Bag set to use tracking
myTransitBag				:= 0;//Transit position	optional
bufferSettleTime			:= 300;  	// Time for bag to settle at buffer in.

//Vars for myOutBag, bufferclear and bagarrived MUST be set in the cyclic task if using request/enable

END_PROGRAM
PROGRAM _CYCLIC
// Set constant LOCAL_MAX_DESTS in local var declaration.

//Inputs
i_bagAtBuffer				:= X[myIO].X02;
//i_bagAtBuffer				:= RequestRel.IC[1];

i_bagAtBufferOut[1] 		:= FALSE; // Any Single bag buffer out IO.
i_bufferOutOpen[1]			:= FALSE;
i_bagAtBufferOut[2] 		:= FALSE;
i_bufferOutOpen[2]			:= FALSE;

RequestRel.PN[myPoint] 		:= FALSE;

IF (myBag = 0) THEN
	Alarm[mySeq].Bag	:= mySeq + 10000;
ELSE
	Alarm[mySeq].Bag	:= myBag;
END_IF;

Alarm[mySeq].Name 		:= 0;
Alarm[mySeq].Beacon	:= TRUE;
Alarm[mySeq].Extra		:= 0;
Alarm[mySeq].Time		:= 3000;

FOR n := 1 TO no_RecieveLines DO
	bufferClear[n] := Line[myRelLine[n]].Clear AND NOT i_bagAtBufferOut[n] AND NOT i_bufferOutOpen[n];
	bagArrived[n] := bufferClear[n]; // Bag arrived condition here is the same. if we are using request/enable we must override below.
	myOutBag[n] := Line[myRelLine[n]].LastBag;
	o_select[n]	:= FALSE;

	IF (myRelLine[n] > 0) AND Line[myRelLine[n]].Trip AND (Alarm[mySeq].Name = 0)  THEN
		Alarm[mySeq].Name := ALM_SWITCH_FAULT;
		Alarm[mySeq].Bag := Line[myRelLine[n]].LastBag;
		Alarm[mySeq].Time := 200;
	END_IF;

END_FOR;

//For Request/Enable overwrite bufferClear and outbags..
myOutBag[1]	:= 205;
myOutBag[2]	:= 206;
// These are the conditions used to say a bag has arrived. Must be spilt from bufferclear so we do not release double bags due to alignment switches etc..
bagArrived[1] := Request.VC_HighLevel[2] AND (Bag[myOutBag[1]].Cat = 0) AND NOT X[33].X05;
bagArrived[2] := Request.VC_HighLevel[1] AND (Bag[myOutBag[2]].Cat = 0) AND NOT X[31].X05;
//Bufferclear. Condition used to check the a buffer is clear for a bag to be released to. Check conditional things here, like safety stops and recieve switches on vc's
bufferClear[1] := bagArrived[1] AND Y[34].Y05 ; // Y[32].Y05 is safety stop we put this in the buffer clear condition only so we do not release a double bag if the recieve switch fails.
bufferClear[2] := bagArrived[2] AND Y[32].Y05;

o_reset			:= FALSE;
o_openBuffer	:= FALSE;

//Setup Sequence
step := D[900 + mySeq];
//Setup Pulse contact
pls := (step <> lastStep);
lastStep := step;

//Sequence
IF (step = 0) THEN
	//Disabled
END_IF;

//_reset Points
ton_10ms_reset(IN:=((step = 1) AND NOT Std.HaltSysZone[myZone]), PT:= 200);
IF (step = 1) THEN
	o_reset := NOT Std.HaltSysZone[myZone];
	IF ton_10ms_reset.Q THEN
		D[900 + mySeq] := 2;
		Count[mySeq] := Count[mySeq] + 1;
	END_IF;
END_IF;

//Wait for bag to settle at buffer
ton_10ms_SettledBuffer(IN:= i_bagAtBuffer, PT:= bufferSettleTime);
IF (step = 2) THEN
	IF ton_10ms_SettledBuffer.Q AND NOT Std.HaltSysZone[myZone] THEN
		IF (alt >= no_RecieveLines) THEN
			alt := 1;
		ELSE
			alt := alt + 1;
		END_IF;
		IF (myBag > 0) THEN // Full
			IF (Bag[myBag].Cat > 0) THEN
				RequestRel.PN[myPoint] := 1;
				myLine :=  0;
				//	Decide which line the bag is going to.
				IF useDestinations THEN
					FOR n := 1 TO no_RecieveLines DO // Search FOR the buffer with matching destination
						FOR x := 1 TO LOCAL_MAX_DESTS DO
							IF (myRelLineDest[n].dest[x] = 0) THEN
								myRelLineDest[n].dest[x] := myRelLine[n];
							END_IF;
							IF Bag[myBag].Dst = myRelLineDest[n].dest[x] THEN
								myLine := n;
							END_IF;
							IF (myLine > 0)THEN
								EXIT;
							END_IF;
						END_FOR;
						IF (myLine > 0) THEN
							EXIT;
						END_IF;
					END_FOR;
				ELSE
					myLine := alt;
				END_IF;
				//Check data valid
				IF (myLine > 0) AND (myLine <= LOCAL_MAX_DESTS) THEN
					IF (myTransitBag > 0)  AND (myOutBag[myLine] > 0) THEN
						IF bufferClear[myLine] AND (Bag[myOutBag[myLine]].Cat = 0) AND (Bag[myTransitBag].Cat = 0) THEN
							IF (myRelLine[myLine] > 0) THEN
								C[myRelLine[myLine]] := 0;
							END_IF;
							Bag[myTransitBag] := Bag[myBag];
							Bag[myBag] := Bag[0];
							D[900 + mySeq] := step + myLine;
						ELSIF (Bag[myTransitBag].Cat > 0) THEN
							Alarm[mySeq].Name := ALM_BAG_DATA_ERROR;
							Alarm[mySeq].Bag := myTransitBag;
						ELSIF Line[myRelLine[myLine]].Clear THEN
							Alarm[mySeq].Name := ALM_BAG_NOT_SHOWN_ON_SCREEN;
							Alarm[mySeq].Bag := myOutBag[myLine];
						END_IF;
					ELSIF (myOutBag[myLine] > 0) THEN // Don;t use tranit bag.
						IF bufferClear[myLine] AND (Bag[myOutBag[myLine]].Cat = 0) THEN
							IF (myRelLine[myLine] > 0) THEN
								C[myRelLine[myLine]] := 0;
							END_IF;
							D[900 + mySeq] := step + myLine;
						ELSIF Line[myRelLine[myLine]].Clear THEN
							Alarm[mySeq].Name := ALM_BAG_NOT_SHOWN_ON_SCREEN;
							Alarm[mySeq].Bag := myOutBag[myLine];
						END_IF;
					ELSE//Not configured correctly...
						Alarm[mySeq].Name := ALM_GENERAL_SEQUENCE;
					END_IF;
				ELSE
					Alarm[mySeq].Name := ALM_DEST_NOT_VALID;
				END_IF;
			ELSIF (Bag[myBag].Cat = 0) THEN
				Alarm[mySeq].Name := ALM_BAG_DATA_ERROR;
			END_IF;
		ELSE
			//Empty Bag
			RequestRel.PN[myPoint] := 1;
			IF bufferClear[alt] THEN
				IF (myRelLine[alt] > 0) THEN
					C[myRelLine[alt]] := 0;
				END_IF;
				D[900 + mySeq] := step + alt;
			END_IF;
		END_IF;
	ELSIF ((myBag > 0) AND (Bag[myBag].Cat > 0) AND NOT i_bagAtBuffer AND NOT Std.HaltSysZone[myZone]) THEN
		Alarm[mySeq].Name := ALM_BAG_NOT_SETTLED;
	END_IF;
END_IF;

//Select Points AND release bag,NOTE step is greater than OR equal TO 3 so it will be a different step number FOR each destination.
IF (step >= 3) THEN
	myLine := step - 2;
	releaseValid := ((myTransitBag = 0) OR ((Bag[myTransitBag].Cat > 0) AND (Bag[myOutBag[myLine]].Cat = 0)));
	o_select[myLine] :=	TRUE;
	o_openBuffer := releaseValid;
	bagReleased := (((myRelLine[myLine] > 0) AND Line[myRelLine[myLine]].Trip) OR ((myRelLine[myLine] = 0) AND NOT bagArrived[myLine]));
	IF bagReleased AND releaseValid THEN
		IF (myTransitBag > 0) AND (myOutBag[myLine] > 0) AND (myRelLine[myLine] > 0) THEN//Only transfer bag data out when releasing to a buffer.
			Bag[myOutBag[myLine]] := Bag[myTransitBag];
			Bag[myTransitBag] := Bag[0];
		ELSIF (myTransitBag = 0) AND (myOutBag[myLine] > 0) AND (myRelLine[myLine] > 0) THEN//Only transfer bag data out when releasing to a buffer.
			Bag[myOutBag[myLine]] := Bag[myBag];
			Bag[myBag] := Bag[0];
		END_IF;
		IF (myRelLine[myLine] = 0) AND (myBag > 0) THEN // Check data has been deleted by outgoing sequence when tracking bags and using request/enable
			IF Bag[myTransitBag].Cat = 0 THEN
				D[900 + mySeq]  := 1;
			ELSE
				Alarm[mySeq].Name := ALM_BAG_DATA_ERROR;
			END_IF;
		ELSE
			D[900 + mySeq]  := 1;
		END_IF;
	ELSIF NOT releaseValid THEN
		IF Bag[myTransitBag].Cat = 0 THEN
			Alarm[mySeq].Name := ALM_BAG_DATA_ERROR;
		ELSIF Line[myRelLine[myLine]].Clear AND (Bag[myOutBag[myLine]].Cat > 0) THEN
			Alarm[mySeq].Name := ALM_BAG_DATA_ERROR;
			Alarm[mySeq].Bag := myOutBag[myLine];
		END_IF;
	ELSIF releaseValid AND (myRelLine[myLine] > 0) THEN
		Alarm[mySeq].Name := ALM_BAG_NOT_RELEASED;
		Alarm[mySeq].Time := 1500;
	END_IF;
END_IF;

//-----------------------------------
//PLC Outputs - adjust TO suit system
//-----------------------------------

Y[myIO].Y06 := o_openBuffer;
//EnableRel.IC[1] := o_openBuffer;// Example of using RequestRel interface.

Y[myIO].Y07 := o_select[1];
Y[myIO].Y08 := o_reset OR o_select[2];

//Alarms
timerAlarm(IN := NOT pls AND (Alarm[mySeq].Name > 0),PT:= Alarm[mySeq].Time);

Alarm[mySeq].On 	:= timerAlarm.Q;
Alarm[mySeq].ET 	:= timerAlarm.ET;

END_PROGRAM
```

### Program Logical/BaseStandards/Points/ComplexPoints/x_1_Point (IEC, version 2.00.6) - *Standard Point multi lines into 1

#### x_1_Point.st - Implementation code
```iecst
(********************************************************************
 * COPYRIGHT --
 ********************************************************************
 * PROGRAM: x_1_Point
 * File: x_1_Point.st
 * Author: treamsbottom
 * Created: July 9, 2015
 ********************************************************************
 * Implementation OF PROGRAM x_1_Point
 ********************************************************************)
// V1 - 09 July 2015 T.R First Release
//V2.00.1 First release compliant with new standards.
//V2.00.2 Add Destination Valid check, Only release a bag when it has a valid destination.
//V2.00.3 Add Buffer out position.. A fake bag register for outgoing sequences to check for data valid before enabling..
//V2.00.4 Make Transit bag optional

PROGRAM _INIT
// Configuration

//SET LOCAL_MAX_BUFFERS to set number of buffers..
	mySeq				:= 14;	//Sequence number

	myRelLine			:= 45; 	// Set TO 0 TO use request....
	myPoint				:= 7;

	myZone				:= 1;
	myIO				:= 107;

	useDestinations		:= 0; // Set to true to wait for a destination to be valid before going into the buffer queue. NB> This does not alarm as it only expected to work with a search function.

	myBag[1]			:= 305; // Buffer Bags
	myBag[2]			:= 301;

	myTransitBag		:= 0; // Set to use transit bag before out bag..
	mySelectedBag		:= 0; // A bag to show to the next sequence which bag has been selected. USE INSTEAD OF myTransitBag

	FOR n := 1 TO LOCAL_MAX_BUFFERS DO
		bufferSettleTime[n] := 300;
	END_FOR;

	IF (myRelLine > 0) THEN
		myOutBag		:= Line[myRelLine].LastBag;
	ELSE
		myOutBag 		:= 0; //Set bag number here if using request/enable AND tracking....
	END_IF;

END_PROGRAM

PROGRAM _CYCLIC

	i_bagAtBuffer[1]	:= X[myIO].X01;	//Set request release here if required
	i_bagAtBuffer[2]	:= X[myIO].X02;

	i_bagAtBufferOut 	:= FALSE;
	i_bufferOutOpen		:= FALSE;

	o_reset				:= FALSE;

	FOR n := 0 TO LOCAL_MAX_BUFFERS DO
		o_openBuffer[n]	:= FALSE;
		o_select[n]		:= FALSE;
	END_FOR;

	Request.PN[myPoint] := FALSE;
	RequestRel.PN[myPoint] := FALSE;

	Bag[mySelectedBag] := Bag[0];

	IF myOutBag = 0 THEN
		Alarm[mySeq].Bag	:= mySeq + 10000;
		myTransitBag := 0; // If out bag is not defined we cannot track bags do delete mapping of transit bag.
	ELSE
		Alarm[mySeq].Bag	:= myOutBag;
	END_IF;

	Alarm[mySeq].Name 	:= 0;
	Alarm[mySeq].Beacon	:= TRUE;
	Alarm[mySeq].Extra	:= 0;
	Alarm[mySeq].Time	:= 3000;

	//Setup Sequence
	step := D[900 + mySeq];
	//Setup Pulse contact
	pls := (step <> laststep);
	laststep := step;

	//Sequence
	IF (step = 0) THEN
		//Disabled
	END_IF;

	//Reset Points

	ton_10ms_reset(IN:=((step = 1) AND NOT Std.HaltSysZone[myZone]), PT:= 200);
	IF (step = 1) THEN
		o_reset := NOT Std.HaltSysZone[myZone];
		IF ton_10ms_reset.Q THEN
			D[900 + mySeq] := 2;
			Count[mySeq] := Count[mySeq] + 1;
		END_IF;
	END_IF;

	FOR n := 1 TO LOCAL_MAX_BUFFERS DO
		ton_10ms_settledbuffer[n](IN := i_bagAtBuffer[n],PT := bufferSettleTime[n]);
		IF (myBag[n] > 0) THEN // Bag tracking
			IF useDestinations THEN
				myDest := Bag[myBag[n]].Dst;
				IF (myDest > 0) AND (myDest <= MAX_DESTINATIONS) THEN
					destValid :=  (Line[myDest].Space > 0) AND Line[myDest].Clear;
				ELSE
					destValid := FALSE;
				END_IF;
			ELSE
				destValid := TRUE;
			END_IF;

			lineValid[n] := ton_10ms_settledbuffer[n].Q AND (Bag[myBag[n]].Cat > 0);

			IF ton_10ms_settledbuffer[n].Q AND (Bag[myBag[n]].Cat = 0) THEN
				Alarm[mySeq].Name := ALM_BAG_DATA_ERROR;
				Alarm[mySeq].Bag := myBag[n];
			END_IF;
		ELSE
			destValid := 1;
			lineValid[n] := ton_10ms_settledbuffer[n].Q;
		END_IF;
		IF lineValid[n] AND destValid THEN
			IF (waitTime[n] < 16#FFFFFFFF) THEN
				waitTime[n]:= waitTime[n] + 1;
			END_IF;
		ELSE
			waitTime[n] := 0;
		END_IF;
	END_FOR;

	waitingLongest := 0;
	waitTime[0] := 0;
	FOR n := 1 TO LOCAL_MAX_BUFFERS DO
		IF waitTime[n] > waitTime[0] THEN
			waitTime[0] := waitTime[n];
			waitingLongest := n;
		END_IF;
	END_FOR;

	IF (myRelLine > 0) THEN
		IF (myTransitBag > 0) THEN
			bufferClear := Line[myRelLine].Clear AND (Bag[myOutBag].Cat = 0) AND (Bag[myTransitBag].Cat = 0) AND NOT i_bagAtBufferOut AND NOT i_bufferOutOpen;
		ELSIF (myOutBag > 0) THEN
			bufferClear := Line[myRelLine].Clear AND (Bag[myOutBag].Cat = 0) AND NOT i_bagAtBufferOut AND NOT i_bufferOutOpen;
		ELSE
			bufferClear := Line[myRelLine].Clear AND NOT i_bagAtBufferOut AND NOT i_bufferOutOpen;
		END_IF;
	ELSE // Wait FOR enable Release
		IF (mySelectedBag > 0) THEN // Check data has been copied out by enabling sequence.
			bufferClear := EnableRel.PN[myPoint] AND (Bag[myOutBag].Cat > 0) AND NOT i_bagAtBufferOut AND NOT i_bufferOutOpen;
		ELSIF (myTransitBag > 0) THEN
			bufferClear := EnableRel.PN[myPoint] AND (Bag[myOutBag].Cat = 0) AND (Bag[myTransitBag].Cat = 0) AND NOT i_bagAtBufferOut AND NOT i_bufferOutOpen;
		ELSIF (myOutBag > 0) THEN
			bufferClear := EnableRel.PN[myPoint] AND (Bag[myOutBag].Cat = 0) AND NOT i_bagAtBufferOut AND NOT i_bufferOutOpen;
		ELSE
			bufferClear := EnableRel.PN[myPoint] AND NOT i_bagAtBufferOut AND NOT i_bufferOutOpen;
		END_IF;
	END_IF;

	IF (step = 2) THEN
		IF (waitingLongest <= LOCAL_MAX_BUFFERS) THEN // Keep arrays in range
			RequestRel.PN[myPoint] := (waitingLongest > 0) AND (myRelLine = 0); // Request release if a buffer is waiting to release.
			IF (mySelectedBag > 0) AND (waitingLongest > 0) THEN
				Bag[mySelectedBag] := Bag[myBag[waitingLongest]];
			END_IF;
			IF bufferClear AND lineValid[waitingLongest] AND NOT Std.HaltSysZone[myZone] THEN
				IF (myBag[waitingLongest] > 0) THEN
					IF (myTransitBag > 0) THEN// Copy data to transit position
						Bag[myTransitBag] := Bag[myBag[waitingLongest]];
						Bag[myBag[waitingLongest]] := Bag[0];
					ELSIF (mySelectedBag > 0) THEN
						Bag[myBag[waitingLongest]] := Bag[0];
					END_IF;
				END_IF;
				IF (myRelLine > 0) THEN
					C[myRelLine] := 0;
				END_IF;
				D[900 + mySeq] := step + waitingLongest;
			ELSIF (myTransitBag > 0) AND (Bag[myTransitBag].Cat > 0) THEN
				Alarm[mySeq].Name := ALM_BAG_DATA_ERROR;
				Alarm[mySeq].Bag := myTransitBag;
			ELSIF (myOutBag > 0) AND Line[myRelLine].Clear AND (Bag[myOutBag].Cat > 0) THEN
				Alarm[mySeq].Name := ALM_BAG_DATA_ERROR;
			END_IF;
		ELSE
			Alarm[mySeq].Name := ALM_GENERAL_SEQUENCE;
		END_IF;
	END_IF;

	//Select Points AND release bag,NOTE step is greater than OR equal TO 3 so it will be a different step number FOR each destination.
	IF (step >= 3) THEN
		myLine := step - 2;
		releaseValid := ((mySelectedBag > 0) OR (myOutBag = 0) OR ((myTransitBag > 0) AND (Bag[myOutBag].Cat = 0) AND (Bag[myTransitBag].Cat > 0))
		OR ((myOutBag > 0) AND  (myTransitBag = 0)  AND (Bag[myOutBag].Cat = 0) AND (Bag[myBag[myLine]].Cat > 0)));
		o_select[myLine] :=	TRUE;
		o_openBuffer[myLine] := releaseValid;
		bagArrived := (((myRelLine > 0) AND Line[myRelLine].Trip) OR ((myRelLine = 0) AND NOT EnableRel.PN[myPoint]));
		IF bagArrived AND releaseValid THEN
			IF (myTransitBag > 0) AND (myRelLine > 0) THEN//Only copy data out if not using RequestRel
				Bag[myOutBag] := Bag[myTransitBag];
				Bag[myTransitBag] := Bag[0];
			ELSIF (myOutBag > 0 AND myRelLine > 0) THEN
				Bag[myOutBag] := Bag[myBag[myLine]];
				Bag[myBag[myLine]] := Bag[0];
			END_IF;
			IF (myRelLine = 0) AND (myOutBag > 0) THEN // If using request and tracking make sure data has been deleted from transit bag or outgoing bag. by the enabling sequence
				IF (mySelectedBag > 0) THEN
					IF (Bag[myOutBag].Cat = 0) THEN
						D[900 + mySeq]  := 1;
					END_IF;
				ELSIF (myTransitBag > 0) THEN
					IF (Bag[myTransitBag].Cat = 0) THEN	// Transit bag should
						D[900 + mySeq]  := 1;
					ELSE
						Alarm[mySeq].Time := 0;
						Alarm[mySeq].Bag := myTransitBag;
						Alarm[mySeq].Name := ALM_BAG_DATA_ERROR;
					END_IF;
				ELSE
					IF ((Bag[myOutBag].Cat = 0) AND (Bag[myBag[myLine]].Cat > 0)) THEN
						Bag[myOutBag] := Bag[myBag[myLine]];
						Bag[myBag[myLine]] := Bag[0];
						D[900 + mySeq]  := 1;
					END_IF;
				END_IF;
			ELSE
				D[900 + mySeq] := 1;
			END_IF;
		ELSIF NOT releaseValid THEN
			IF Bag[myOutBag].Cat = 0 THEN
				Alarm[mySeq].Name := ALM_BAG_DATA_ERROR;
			ELSIF Line[myRelLine].Clear AND (Bag[myOutBag].Cat > 0) THEN
				Alarm[mySeq].Name := ALM_BAG_DATA_ERROR;
				Alarm[mySeq].Bag := myOutBag;
			END_IF;
		END_IF;
	END_IF;

	//-----------------------------------
	//PLC Outputs - adjust TO suit system
	//-----------------------------------

	Y[myIO].Y05 := o_openBuffer[1];
	Y[myIO].Y06 := o_openBuffer[2];
	//EnableRel.VC_HighLevel[2] := o_openBuffer[1];// Example of using RequestRel interface.
	//EnableRel.VC_HighLevel[1] := o_openBuffer[2];// Example of using RequestRel interface.

	Y[myIO].Y07 := o_select[1];
	Y[myIO].Y08 := o_reset OR o_select[2];

	//Alarms
	timerAlarm(IN := NOT pls AND (Alarm[mySeq].Name > 0),PT:= Alarm[mySeq].Time);

	Alarm[mySeq].On 	:= timerAlarm.Q;
	Alarm[mySeq].ET 	:= timerAlarm.ET;

END_PROGRAM
```

#### x_1_Point.var - Local variables
```iecst
(********************************************************************
 * COPYRIGHT --
 ********************************************************************
 * Program: x_1_Point
 * File: x_1_Point.var
 * Author: treamsbottom
 * Created: July 9, 2015
 ********************************************************************
 * Local variables of program x_1_Point
 ********************************************************************)
VAR CONSTANT
	LOCAL_MAX_BUFFERS : UINT := 2;
END_VAR
VAR
	mySeq : UINT;
	myRelLine : UINT;
	myPoint : UINT;
	myZone : UINT;
	myIO : UINT;
	myBag : ARRAY[0..LOCAL_MAX_BUFFERS] OF UINT;
	i_bagAtBuffer : ARRAY[0..LOCAL_MAX_BUFFERS] OF BOOL;
	i_bagAtBufferOut : BOOL;
	i_bufferOutOpen : BOOL;
	myOutBag : UINT;
	o_reset : BOOL;
	n : UINT;
	o_openBuffer : ARRAY[0..LOCAL_MAX_BUFFERS] OF BOOL;
	o_select : ARRAY[0..LOCAL_MAX_BUFFERS] OF BOOL;
	step : UINT;
	ton_10ms_reset : TON_10ms;
	pls : BOOL;
	laststep : UINT;
	ton_10ms_settledbuffer : ARRAY[0..LOCAL_MAX_BUFFERS] OF TON_10ms;
	lineValid : ARRAY[0..LOCAL_MAX_BUFFERS] OF BOOL;
	waitTime : ARRAY[0..LOCAL_MAX_BUFFERS] OF UDINT;
	timerAlarm : TON_10ms;
	waitingLongest : UINT;
	bufferClear : BOOL;
	myLine : UINT;
	releaseValid : BOOL;
	bagArrived : BOOL;
	bufferSettleTime : ARRAY[0..LOCAL_MAX_BUFFERS] OF UDINT;
	useDestinations : BOOL;
	mySelectedBag : UINT;
	myDest : UINT;
	myTransitBag : UINT;
	destValid : BOOL;
END_VAR
```

### Program Logical/BaseStandards/Points/ComplexPoints/x_x_Point (IEC, version 1.00.1) - *Standard point for many to many MAX 9 buffer & MAX 9 Lines

#### x_x_point.st - Implementation code
```iecst
(********************************************************************
* COPYRIGHT --
********************************************************************
* Program: pr
* File: pr.st
* Author: treamsbottom
* Created: July 16, 2015
********************************************************************
* Implementation of program Point x_x
********************************************************************)
// LIMITS CAN ONLY 9 BUFFERS AND 9 RELEASE LINES!!//
//V1.00.1 First Release

PROGRAM _INIT
//Configuration
mySeq						:= 24;	//Sequence number
myIO						:= 103;
myZone						:= 0;
myRelLine[1]				:= 25;
myRelLine[2]				:= 12;

myBuffBag[1]				:= 326;
myBuffBag[2]				:= 125;

//Configure the destination Maps for each release line
destCheck[1].Dests[1] := 25;// Line 1 can only recieve bags with of 25

destCheck[2].Dests[1] := EMPTY_BAG;// relLine 2 can recieve bags empty bags or bags for dischager 6. // Destination of 0 is valid.
destCheck[2].Dests[2] := 26;//

FOR line := 1 TO MAX_LINES_OUT DO
	myOutBag[line] 			:= Line[myRelLine[line]].LastBag;
END_FOR;

bufferSettleTime			:= 300;

alarm						ACCESS ADR(Alarm[mySeq]);

END_PROGRAM

PROGRAM _CYCLIC
//Inputs
i_bagAtBuffer[1]			:= X[myIO].X01;
i_bagAtBuffer[2]			:= X[myIO].X02;

i_bagAtBufferOut[1] 	:= FALSE; // Any Single bag buffer out IO.
i_bufferOutOpen[1]		:= FALSE;
i_bagAtBufferOut[2] 	:= X[105].X01;
i_bufferOutOpen[2]		:= Y[105].Y05;

o_reset					:= FALSE;
FOR buffer := 1 TO MAX_LINES_IN DO
	o_openBuffer[buffer]			:= FALSE;
	queue.input[buffer] 			:= i_bagAtBuffer[buffer]; //Input for buffer queues..
END_FOR;

FOR line := 1 TO MAX_LINES_OUT DO
	o_select[line]			:= FALSE;
	IF (myRelLine[line] > 0) THEN
		lineReadyToRecieve[line] := (Line[myRelLine[line]].Clear AND ((Bag[myOutBag[line]].Cat = 0) OR (myOutBag[line] = 0)) AND NOT i_bagAtBufferOut[line] AND NOT i_bufferOutOpen[line]);
		lineBagRecieved[line] := Line[myRelLine[line]].Trip;
	END_IF;
END_FOR;
// Set your own conditions here if not using lines
//myOutBag[1] := 0;//
//lineReadyToRecieve[1] := ;//This is used to check if we can release to the line, so we can check things like rail align sensors..
//lineBagRecieved[line] := ;//This is condition for when the bag has arrived..

IF (myBuffBag[1] = 0) THEN
	alarm.Bag	:= mySeq + 10000;
ELSE
	alarm.Bag	:= myBuffBag[1];
END_IF;

alarm.Name 		:= 0;
alarm.Beacon	:= TRUE;
alarm.Extra		:= 0;
alarm.Time		:= 3000;

//Setup Sequence
step := D[900 + mySeq];
//Setup Pulse contact
pls := (step <> lastStep);
lastStep := step;

//Sequence
IF (step = 0) THEN
	//Disabled
END_IF;

IF (step > 0) THEN
	_alarms;
END_IF;
//step 1 reset points
ton_reset(IN:= (step = 1),PT:= 300);
IF (step = 1) THEN
	o_reset := 1;
	IF ton_reset.Q AND NOT Std.HaltSysZone[myZone] THEN
		D[900 + mySeq] := 2;
	END_IF;
END_IF;

//Step 2 choose which bag has been waiting longest and decide where to send it.
//Inputs in loop above //
queue.settleTime 	:= bufferSettleTime;
FOR line := 1 TO MAX_LINES_OUT DO
	destQueue.input[line] := lineReadyToRecieve[line];
END_FOR;
destQueue.settleTime := 10;

IF (step = 2) THEN
	IF NOT Std.HaltSysZone[myZone] THEN
		IF (queue.waitingLongest > 0) THEN
			buffer := queue.waitingLongest;
			line := destQueue.waitingLongest;
			bag_buff		ACCESS ADR(Bag[myBuffBag[buffer]]);	 // Always set the references.. Even if the ref is to 0. Will cause PLC to fail if pointer is not valid.
			//Tracking bags.
			IF (myBuffBag[buffer] > 0) THEN
				//First check if we have Valid data.. If not reset the queue time.
				IF (bag_buff.Cat > 0) THEN
					// We need to check if a destination has to be set and is vaild.
					IF lineReadyToRecieve[line] THEN // First check the buffer that has been waiting longest.
						FOR d := 1 TO MAX_LINES_OUT DO
							IF ((bag_buff.Dst = destCheck[line].Dests[d]) AND  (destCheck[line].Dests[d] > 0)) OR ((bag_buff.Cat = Std.MaxCats) AND (destCheck[line].Dests[d] = EMPTY_BAG)) THEN
								selectedLine := line;
								EXIT;
							END_IF;
						END_FOR;
					END_IF;	//IF no bag found try all the other outgoing buffers
					IF (selectedLine = 0) THEN
						FOR line := 1 TO MAX_LINES_OUT DO
							FOR d := 1 TO MAX_LINES_OUT DO
								IF (lineReadyToRecieve[line] AND (((bag_buff.Dst = destCheck[line].Dests[d]) AND  (destCheck[line].Dests[d] > 0)) OR ((bag_buff.Cat = Std.MaxCats) AND (destCheck[line].Dests[d] = EMPTY_BAG))))  THEN
									selectedLine := line;
									EXIT;
								END_IF;
							END_FOR;
							IF (selectedLine > 0) THEN EXIT; END_IF;
						END_FOR;
					END_IF;
				END_IF;
				IF (selectedLine = 0) THEN // No line has been found so remove it from the queue to search the other lines.
					queue.input[buffer] := FALSE;//<-- Problem here is that we reset the settle time!!!
				END_IF;
			ELSE // No tracking.
			//	selectedLine := destQueue.waitingLongest;
			END_IF;
			IF (selectedLine > 0) THEN // Go to next step.
				D[900 + mySeq] :=  (buffer * 10) + selectedLine ;
			END_IF;
		END_IF;
		_alarms;
	END_IF;
ELSE
	selectedLine := 0;
END_IF;

//Step (Increments of 10 is the buffer, remain is line to send to)
IF (step >= 11) THEN
	buffer :=  (step / 10);
	line := step MOD 10;
	//Check ranges
	IF (buffer > 0) AND (line > 0) AND (buffer <= MAX_LINES_IN) AND (line <= MAX_LINES_OUT) THEN
		bag_buff		ACCESS ADR(Bag[myBuffBag[buffer]]);
		bag_out		 	ACCESS ADR(Bag[myOutBag[line]]);
		IF lineReadyToRecieve[line] THEN
			IF (myRelLine[line] > 0) THEN
				C[myRelLine[line]] := 0;
			END_IF;
			releaseValid := 1;
		END_IF;
		IF releaseValid THEN
			o_select[line] := 1;
			o_openBuffer[buffer] := 1;
			IF lineBagRecieved[line] THEN
				IF (myOutBag[line] > 0) AND (myBuffBag[buffer] > 0) THEN // Move bag data if required.
					bag_out := bag_buff;
					bag_buff := Bag[0];
				END_IF;
				D[900 + mySeq] := 1;
			ELSE
				alarm.Name := ALM_BAG_NOT_RELEASED;
			END_IF;
		END_IF;
	ELSE
		alarm.Name := ALM_GENERAL_SEQUENCE;
		alarm.Time := 0;
	END_IF;
ELSE
	releaseValid := 0;
END_IF;

queue(); // Function for incoming buffer queue
destQueue(); // Outgoing buffer queue.

//-----------------------------------
//PLC Outputs - adjust TO suit system
//-----------------------------------

Y[myIO].Y05 := o_openBuffer[1];
Y[myIO].Y06 := o_openBuffer[2];

Y[myIO].Y07 := o_openBuffer[1];
Y[myIO].Y08 := o_openBuffer[2] OR o_reset;

Y[myIO + 1].Y07 	:= o_select[1];
Y[myIO + 1].Y08 	:= o_select[2] OR o_reset;

//Alarms
timerAlarm(IN := NOT pls AND (alarm.Name > 0),PT:= alarm.Time);

alarm.On 	:= timerAlarm.Q;
alarm.ET 	:= timerAlarm.ET;

END_PROGRAM
```

#### x_x_point.var - Local variables
```iecst
(********************************************************************
 * COPYRIGHT --
 ********************************************************************
 * Program: pr
 * File: pr.var
 * Author: treamsbottom
 * Created: July 16, 2015
 ********************************************************************
 * Local variables of program pr
 ********************************************************************)
VAR
	destCheck : ARRAY[0..MAX_LINES_IN] OF destCheck_typ;
END_VAR
VAR CONSTANT
	MAX_LINES_IN : USINT := 2;
	MAX_LINES_OUT : USINT := 2;
END_VAR
VAR
	mySeq : UINT;
	myIO : UINT;
	myZone : UINT;
	myRelLine : ARRAY[0..MAX_LINES_OUT] OF UINT;
	i_bagAtBuffer : ARRAY[0..MAX_LINES_IN] OF BOOL;
	i_bagAtBufferOut : ARRAY[0..MAX_LINES_OUT] OF BOOL;
	i_bufferOutOpen : ARRAY[0..MAX_LINES_OUT] OF BOOL;
	o_openBuffer : ARRAY[0..MAX_LINES_IN] OF BOOL;
	step : UINT;
	pls : BOOL;
	timerAlarm : TON_10ms;
END_VAR
VAR RETAIN
	lastStep : UINT;
END_VAR
VAR
	bufferSettleTime : UDINT;
	myOutBag : ARRAY[0..MAX_LINES_OUT] OF UINT;
	myBuffBag : ARRAY[0..MAX_LINES_IN] OF UINT;
	alarm : REFERENCE TO Alm;
	bag : REFERENCE TO Bag_typ;
	bag_buff : REFERENCE TO Bag_typ;
	bag_out : REFERENCE TO Bag_typ;
	line_release : REFERENCE TO Line_Typ;
	queue : getWaitingLongest;
	o_select : ARRAY[0..MAX_LINES_OUT] OF BOOL;
	buffer : UINT;
	o_reset : BOOL;
	ton_reset : TON_10ms;
	n : UINT;
	destQueue : getWaitingLongest;
	lineReadyToRecieve : ARRAY[0..MAX_LINES_OUT] OF BOOL;
	x : UINT;
	d : USINT;
	selectedLine : UINT;
	line : UINT;
END_VAR
VAR CONSTANT
	EMPTY_BAG : USINT := 255; (**Const used to send empty bags to a line when tracking*)
END_VAR
VAR
	lineBagRecieved : ARRAY[0..MAX_LINES_OUT] OF BOOL;
	releaseValid : BOOL;
END_VAR
```

#### x_x_point.typ
```iecst
TYPE
	destCheck_typ : 	STRUCT
		Dests : ARRAY[0..MAX_LINES_OUT]OF USINT; (**bag destinations which can be sent to this line.. 0 is valid.*)
	END_STRUCT;
END_TYPE
```

#### _alarms.st
```iecst
ACTION _alarms:
	// Alarms when tracking bags only
	FOR buffer := 1 TO MAX_LINES_IN DO
		IF (myBuffBag[buffer] > 0) THEN
			bag_buff		ACCESS ADR(Bag[myBuffBag[buffer]]);
			IF (bag_buff.Cat = 0) AND i_bagAtBuffer[buffer] THEN
				alarm.Name := ALM_BAG_DATA_ERROR;
				alarm.Time := 0;
				alarm.Bag := myBuffBag[buffer];
			ELSIF bag_buff.Cat > 0 AND NOT i_bagAtBuffer[buffer] AND (step < 3) THEN
				alarm.Name := ALM_BAG_NOT_SETTLED;
				alarm.Time := bufferSettleTime;
				alarm.Bag := myBuffBag[buffer];
			END_IF;
		END_IF;
	END_FOR;
	//
	FOR line := 1 TO MAX_LINES_OUT DO
		IF (myRelLine[line] > 0) THEN
			bag_out		 	ACCESS ADR(Bag[myOutBag[line]]);
			IF Line[myRelLine[line]].Trip THEN
				alarm.Name := ALM_SWITCH_FAULT;
				alarm.Time := 500;
				alarm.Bag := Line[myRelLine[line]].LastBag;
			ELSIF (myOutBag[line] > 0) THEN
				IF (Line[myRelLine[line]].Clear AND (bag_out.Cat > 0)) OR (Line[myRelLine[line]].Full AND (bag_out.Cat = 0)) THEN
					alarm.Name := ALM_SWITCH_FAULT;
					alarm.Time := 500;
					alarm.Bag := myOutBag[line];
				END_IF;
			END_IF;
		END_IF;
	END_FOR;
END_ACTION
```

### Package Logical/BaseStandards/Pneumatic - Pneumatic VC,Incline

### Program Logical/BaseStandards/Pneumatic/pc (IEC, version 1.00.2) - *Pneumatic VC

- Standard_Sequence_PneumaticVC_V1.00.1_ENG.docx (binary file, 207633 bytes)
